# B&R Automation Studio project NAEUL004C00R13L518F00 (part 34)

#### Act_Background3.st - Do Not Change!!!
```iecst
ACTION Act_Background3: //For BHTC Machines

	IF EDGEPOS(tylocalTLBuz.In.bUIManualMod) THEN

		fbBlink(bEn := FALSE);
		fbWarning(bEn := FALSE);

		tylocalTLBuz.Out.bTLRed		:= FALSE;
		tylocalTLBuz.Out.bTLAmber	:= TRUE;
		tylocalTLBuz.Out.bTLGreen	:= FALSE;
		tylocalTLBuz.Out.bBuzBeep	:= FALSE;

	ELSIF tylocalTLBuz.In.bUIManualMod THEN

		IF tylocalTLBuz.In.bErr = TRUE THEN

			fbBlink.tOnTm	:= tylocalTLBuz.In.tTLErrBlinkTm; //Error T#500ms (from NtParam)
			fbBlink.tOffTm	:= tylocalTLBuz.In.tTLErrBlinkTm; //Error T#500ms (from NtParam)

			fbWarning.tOnTm					:= tylocalTLBuz.In.tBuzErrOnTm; //Warn T#500ms (from NtParam)
			fbWarning.tOffTm				:= tylocalTLBuz.In.tBuzErrOnTm; //Warn T#500ms (from NtParam)
			fbWarning.tRstTm				:= tylocalTLBuz.In.tBuzErrRestTm; //Rest 5 seconds (from NtParam)
			fbWarning.usiOnCnt				:= tylocalTLBuz.In.usiBuzErrOnCntr; //Count 3 times (from NtParam)
			fbWarning.bStopAftRptSeqEn		:= tylocalTLBuz.In.bBuzErrStopSeqEn; //Enable Sequence Count (from NtParam)
			fbWarning.usiStopAftRptSeqCntr	:= tylocalTLBuz.In.usiBuzErrStopSeqCntr; //Sequence Counter  (from NtParam)

			fbBlink(bEn := TRUE);
			fbWarning(bEn := TRUE);

			tylocalTLBuz.Out.bTLAmber	:= fbBlink.bOut;
			tylocalTLBuz.Out.bBuzBeep	:= (fbWarning.bOut) AND (tylocalTLBuz.In.bMuteBuz = FALSE);

			bManualErrOn := TRUE;

		ELSIF bManualErrOn THEN

			fbBlink(bEn := FALSE);
			fbWarning(bEn := FALSE);

			tylocalTLBuz.Out.bTLAmber	:= FALSE;
			tylocalTLBuz.Out.bBuzBeep	:= FALSE;

			bManualErrOn := FALSE;

		END_IF

	ELSIF tylocalTLBuz.In.bUIManualMod = FALSE THEN

		bManualErrOn := FALSE;

		IF tylocalTLBuz.In.bStartup = TRUE THEN //Startup, 3 colour ON

			fbBlink(bEn := FALSE);
			fbWarning(bEn := FALSE);

			tylocalTLBuz.Out.bTLBlue		:= TRUE;
			tylocalTLBuz.Out.bTLAmber	:= TRUE;
			tylocalTLBuz.Out.bTLWhite	:= TRUE;
			tylocalTLBuz.Out.bTLGreen	:= TRUE;
			tylocalTLBuz.Out.bBuzBeep	:= FALSE;

		ELSIF tylocalTLBuz.In.bErr = TRUE THEN //Machine Error,Green TL Off, Red TL Blink

			fbBlink.tOnTm	:= tylocalTLBuz.In.tTLErrBlinkTm; //Error T#500ms (from NtParam)
			fbBlink.tOffTm	:= tylocalTLBuz.In.tTLErrBlinkTm; //Error T#500ms (from NtParam)

			fbWarning.tOnTm					:= tylocalTLBuz.In.tBuzErrOnTm; //Warn T#500ms (from NtParam)
			fbWarning.tOffTm				:= tylocalTLBuz.In.tBuzErrOnTm; //Warn T#500ms (from NtParam)
			fbWarning.tRstTm				:= tylocalTLBuz.In.tBuzErrRestTm; //Rest 5 seconds (from NtParam)
			fbWarning.usiOnCnt				:= tylocalTLBuz.In.usiBuzErrOnCntr; //Count 3 times (from NtParam)
			fbWarning.bStopAftRptSeqEn		:= tylocalTLBuz.In.bBuzErrStopSeqEn; //Enable Sequence Count (from NtParam)
			fbWarning.usiStopAftRptSeqCntr	:= tylocalTLBuz.In.usiBuzErrStopSeqCntr; //Sequence Counter  (from NtParam)

			fbBlink(bEn := TRUE);
			fbWarning(bEn := TRUE);

			tylocalTLBuz.Out.bTLBlue		:= FALSE;
			tylocalTLBuz.Out.bTLAmber	:= fbBlink.bOut;
			tylocalTLBuz.Out.bTLWhite	:= FALSE;
			tylocalTLBuz.Out.bTLGreen	:= FALSE;
			tylocalTLBuz.Out.bBuzBeep	:= fbWarning.bOut AND (tylocalTLBuz.In.bMuteBuz = FALSE);

		ELSIF tylocalTLBuz.In.bErrNoBuz = TRUE THEN //not used (Machine Error With No Buz)

			fbBlink.tOnTm	:= tylocalTLBuz.In.tTLErrBlinkTm; //Error T#500ms, not used (from NtParam)
			fbBlink.tOffTm	:= tylocalTLBuz.In.tTLErrBlinkTm; //Error T#500ms, not used (from NtParam)
			fbBlink(bEn := TRUE);
			fbWarning(bEn := FALSE);

			tylocalTLBuz.Out.bTLBlue		:= FALSE;
			tylocalTLBuz.Out.bTLAmber	:= fbBlink.bOut;
			tylocalTLBuz.Out.bTLWhite	:= FALSE;
			tylocalTLBuz.Out.bTLGreen	:= FALSE;
			tylocalTLBuz.Out.bBuzBeep	:= FALSE;

		ELSIF tylocalTLBuz.In.bWarning[0] = TRUE THEN //Warning or AlarmInfo; [Put Conditions in Act_Link.st]

			fbBlink.tOnTm	:= tylocalTLBuz.In.tTLWarnBlinkTm[0]; //Warn T#500ms (from NtParam)
			fbBlink.tOffTm	:= tylocalTLBuz.In.tTLWarnBlinkTm[0]; //Warn T#500ms (from NtParam)

			fbWarning.tOnTm					:= tylocalTLBuz.In.tBuzWarnOnTm[0]; //Warn T#500ms (from NtParam)
			fbWarning.tOffTm				:= tylocalTLBuz.In.tBuzWarnOnTm[0]; //Warn T#500ms (from NtParam)
			fbWarning.tRstTm				:= tylocalTLBuz.In.tBuzWarnRestTm[0]; //Rest 5 seconds (from NtParam)
			fbWarning.usiOnCnt				:= tylocalTLBuz.In.usiBuzWarnOnCntr[0]; //Count 3 times (from NtParam)
			fbWarning.bStopAftRptSeqEn		:= tylocalTLBuz.In.bBuzWarnStopSeqEn[0]; //Enable Sequence Count (from NtParam)
			fbWarning.usiStopAftRptSeqCntr	:= tylocalTLBuz.In.usiBuzWarnStopSeqCntr[0]; //Sequence Counter  (from NtParam)

			fbBlink(bEn := TRUE);
			fbWarning(bEn := TRUE);

			tylocalTLBuz.Out.bTLBlue		:= FALSE;
			tylocalTLBuz.Out.bTLAmber	:= tylocalTLBuz.In.bStandby; //[tylocalTLBuz.In.bStandby ACCESS p_OpsStatusStop], [p_OpsStatusStop	:= ADR(bStatusStop);]
			tylocalTLBuz.Out.bTLWhite	:= fbBlink.bOut;
			tylocalTLBuz.Out.bTLGreen	:= tylocalTLBuz.In.bOps; //[tylocalTLBuz.In.bOps ACCESS p_OpsStatusRun],  [p_OpsStatusRun	:= ADR(bStatusRun)];
			tylocalTLBuz.Out.bBuzBeep	:= fbWarning.bOut AND (tylocalTLBuz.In.bMuteBuz = FALSE);

		ELSIF tylocalTLBuz.In.bStandby = TRUE THEN //not used

			fbBlink.tOnTm	:= tylocalTLBuz.In.tTLWarnBlinkTm[0];
			fbBlink.tOffTm	:= tylocalTLBuz.In.tTLWarnBlinkTm[0];
			fbBlink(bEn := TRUE);
			fbWarning(bEn := FALSE);

			tylocalTLBuz.Out.bTLBlue		:= FALSE;
			tylocalTLBuz.Out.bTLAmber	:= tylocalTLBuz.In.bStandby;
			tylocalTLBuz.Out.bTLWhite	:= fbBlink.bOut;
			tylocalTLBuz.Out.bTLGreen	:= tylocalTLBuz.In.bOps;
			tylocalTLBuz.Out.bBuzBeep	:= FALSE;

		ELSIF tylocalTLBuz.In.bWarning[1] = TRUE THEN //not used

			fbBlink.tOnTm	:= tylocalTLBuz.In.tTLWarnBlinkTm[1];
			fbBlink.tOffTm	:= tylocalTLBuz.In.tTLWarnBlinkTm[1];

			fbWarning.tOnTm					:= tylocalTLBuz.In.tBuzWarnOnTm[1]; //Warn T#500ms (from NtParam)
			fbWarning.tOffTm				:= tylocalTLBuz.In.tBuzWarnOnTm[1]; //Warn T#500ms (from NtParam)
			fbWarning.tRstTm				:= tylocalTLBuz.In.tBuzWarnRestTm[1]; //Rest 5 seconds (from NtParam)
			fbWarning.usiOnCnt				:= tylocalTLBuz.In.usiBuzWarnOnCntr[1]; //Count 3 times (from NtParam)
			fbWarning.bStopAftRptSeqEn		:= tylocalTLBuz.In.bBuzWarnStopSeqEn[1]; //Enable Sequence Count (from NtParam)
			fbWarning.usiStopAftRptSeqCntr	:= tylocalTLBuz.In.usiBuzWarnStopSeqCntr[1]; //Sequence Counter  (from NtParam)

			fbBlink(bEn := TRUE);
			fbWarning(bEn := TRUE);

			tylocalTLBuz.Out.bTLBlue		:= FALSE;
			tylocalTLBuz.Out.bTLAmber	:= tylocalTLBuz.In.bStandby;
			tylocalTLBuz.Out.bTLWhite	:= fbBlink.bOut;
			tylocalTLBuz.Out.bTLGreen	:= tylocalTLBuz.In.bOps;
			tylocalTLBuz.Out.bBuzBeep	:= fbWarning.bOut AND (tylocalTLBuz.In.bMuteBuz = FALSE);

		ELSIF tylocalTLBuz.In.bWarningNoBuz[1] = TRUE THEN //not used

			fbBlink.tOnTm	:= tylocalTLBuz.In.tTLWarnBlinkTm[1];
			fbBlink.tOffTm	:= tylocalTLBuz.In.tTLWarnBlinkTm[1];
			fbBlink(bEn := TRUE);
			fbWarning(bEn := FALSE);

			tylocalTLBuz.Out.bTLBlue		:= FALSE;
			tylocalTLBuz.Out.bTLAmber	:= tylocalTLBuz.In.bStandby;
			tylocalTLBuz.Out.bTLWhite	:= fbBlink.bOut;
			tylocalTLBuz.Out.bTLGreen	:= tylocalTLBuz.In.bOps;
			tylocalTLBuz.Out.bBuzBeep	:= FALSE;

		ELSIF tylocalTLBuz.In.bWarning[2] = TRUE THEN //not used

			fbBlink.tOnTm	:= tylocalTLBuz.In.tTLWarnBlinkTm[2];
			fbBlink.tOffTm	:= tylocalTLBuz.In.tTLWarnBlinkTm[2];

			fbWarning.tOnTm					:= tylocalTLBuz.In.tBuzWarnOnTm[2]; //Warn T#500ms (from NtParam)
			fbWarning.tOffTm				:= tylocalTLBuz.In.tBuzWarnOnTm[2]; //Warn T#500ms (from NtParam)
			fbWarning.tRstTm				:= tylocalTLBuz.In.tBuzWarnRestTm[2]; //Rest 5 seconds (from NtParam)
			fbWarning.usiOnCnt				:= tylocalTLBuz.In.usiBuzWarnOnCntr[2]; //Count 3 times (from NtParam)
			fbWarning.bStopAftRptSeqEn		:= tylocalTLBuz.In.bBuzWarnStopSeqEn[2]; //Enable Sequence Count (from NtParam)
			fbWarning.usiStopAftRptSeqCntr	:= tylocalTLBuz.In.usiBuzWarnStopSeqCntr[2]; //Sequence Counter  (from NtParam)

			fbBlink(bEn := TRUE);
			fbWarning(bEn := TRUE);

			tylocalTLBuz.Out.bTLBlue	:= FALSE;
			tylocalTLBuz.Out.bTLAmber	:= tylocalTLBuz.In.bStandby;
			tylocalTLBuz.Out.bTLWhite	:= fbBlink.bOut;
			tylocalTLBuz.Out.bTLGreen	:= tylocalTLBuz.In.bOps;
			tylocalTLBuz.Out.bBuzBeep	:= fbWarning.bOut AND (tylocalTLBuz.In.bMuteBuz = FALSE);

		ELSIF tylocalTLBuz.In.bWarningNoBuz[2] = TRUE THEN //not used

			fbBlink.tOnTm	:= tylocalTLBuz.In.tTLWarnBlinkTm[2];
			fbBlink.tOffTm	:= tylocalTLBuz.In.tTLWarnBlinkTm[2];
			fbBlink(bEn := TRUE);
			fbWarning(bEn := FALSE);

			tylocalTLBuz.Out.bTLBlue		:= FALSE;
			tylocalTLBuz.Out.bTLAmber	:= tylocalTLBuz.In.bStandby;
			tylocalTLBuz.Out.bTLWhite	:= fbBlink.bOut;
			tylocalTLBuz.Out.bTLGreen	:= tylocalTLBuz.In.bOps;
			tylocalTLBuz.Out.bBuzBeep	:= FALSE;

		ELSIF tylocalTLBuz.In.bWarning[3] = TRUE THEN //not used

			fbBlink.tOnTm	:= tylocalTLBuz.In.tTLWarnBlinkTm[3];
			fbBlink.tOffTm	:= tylocalTLBuz.In.tTLWarnBlinkTm[3];

			fbWarning.tOnTm					:= tylocalTLBuz.In.tBuzWarnOnTm[3]; //Warn T#500ms (from NtParam)
			fbWarning.tOffTm				:= tylocalTLBuz.In.tBuzWarnOnTm[3]; //Warn T#500ms (from NtParam)
			fbWarning.tRstTm				:= tylocalTLBuz.In.tBuzWarnRestTm[3]; //Rest 5 seconds (from NtParam)
			fbWarning.usiOnCnt				:= tylocalTLBuz.In.usiBuzWarnOnCntr[3]; //Count 3 times (from NtParam)
			fbWarning.bStopAftRptSeqEn		:= tylocalTLBuz.In.bBuzWarnStopSeqEn[3]; //Enable Sequence Count (from NtParam)
			fbWarning.usiStopAftRptSeqCntr	:= tylocalTLBuz.In.usiBuzWarnStopSeqCntr[3]; //Sequence Counter  (from NtParam)

			fbBlink(bEn := TRUE);
			fbWarning(bEn := TRUE);

			tylocalTLBuz.Out.bTLBlue		:= FALSE;
			tylocalTLBuz.Out.bTLAmber	:= tylocalTLBuz.In.bStandby;
			tylocalTLBuz.Out.bTLWhite	:= fbBlink.bOut;
			tylocalTLBuz.Out.bTLGreen	:= tylocalTLBuz.In.bOps;
			tylocalTLBuz.Out.bBuzBeep	:= fbWarning.bOut AND (tylocalTLBuz.In.bMuteBuz = FALSE);

		ELSIF tylocalTLBuz.In.bWarningNoBuz[3] = TRUE THEN //not used

			fbBlink.tOnTm	:= tylocalTLBuz.In.tTLWarnBlinkTm[3];
			fbBlink.tOffTm	:= tylocalTLBuz.In.tTLWarnBlinkTm[3];
			fbBlink(bEn := TRUE);
			fbWarning(bEn := FALSE);

			tylocalTLBuz.Out.bTLBlue		:= FALSE;
			tylocalTLBuz.Out.bTLAmber	:= tylocalTLBuz.In.bStandby;
			tylocalTLBuz.Out.bTLWhite	:= fbBlink.bOut;
			tylocalTLBuz.Out.bTLGreen	:= tylocalTLBuz.In.bOps;
			tylocalTLBuz.Out.bBuzBeep	:= FALSE;

		ELSIF tylocalTLBuz.In.bWarning[4] = TRUE THEN //not used

			fbBlink.tOnTm	:= tylocalTLBuz.In.tTLWarnBlinkTm[4];
			fbBlink.tOffTm	:= tylocalTLBuz.In.tTLWarnBlinkTm[4];

			fbWarning.tOnTm					:= tylocalTLBuz.In.tBuzWarnOnTm[4]; //Warn T#500ms (from NtParam)
			fbWarning.tOffTm				:= tylocalTLBuz.In.tBuzWarnOnTm[4]; //Warn T#500ms (from NtParam)
			fbWarning.tRstTm				:= tylocalTLBuz.In.tBuzWarnRestTm[4]; //Rest 5 seconds (from NtParam)
			fbWarning.usiOnCnt				:= tylocalTLBuz.In.usiBuzWarnOnCntr[4]; //Count 3 times (from NtParam)
			fbWarning.bStopAftRptSeqEn		:= tylocalTLBuz.In.bBuzWarnStopSeqEn[4]; //Enable Sequence Count (from NtParam)
			fbWarning.usiStopAftRptSeqCntr	:= tylocalTLBuz.In.usiBuzWarnStopSeqCntr[4]; //Sequence Counter  (from NtParam)

			fbBlink(bEn := TRUE);
			fbWarning(bEn := TRUE);

			tylocalTLBuz.Out.bTLBlue		:= FALSE;
			tylocalTLBuz.Out.bTLAmber	:= tylocalTLBuz.In.bStandby;
			tylocalTLBuz.Out.bTLWhite	:= fbBlink.bOut;
			tylocalTLBuz.Out.bTLGreen	:= tylocalTLBuz.In.bOps;
			tylocalTLBuz.Out.bBuzBeep	:= fbWarning.bOut AND (tylocalTLBuz.In.bMuteBuz = FALSE);

		ELSIF tylocalTLBuz.In.bWarningNoBuz[4] = TRUE THEN //not used

			fbBlink.tOnTm	:= tylocalTLBuz.In.tTLWarnBlinkTm[4];
			fbBlink.tOffTm	:= tylocalTLBuz.In.tTLWarnBlinkTm[4];
			fbBlink(bEn := TRUE);
			fbWarning(bEn := FALSE);

			tylocalTLBuz.Out.bTLBlue		:= FALSE;
			tylocalTLBuz.Out.bTLAmber	:= tylocalTLBuz.In.bStandby;
			tylocalTLBuz.Out.bTLWhite	:= fbBlink.bOut;
			tylocalTLBuz.Out.bTLGreen	:= tylocalTLBuz.In.bOps;
			tylocalTLBuz.Out.bBuzBeep	:= FALSE;

		ELSIF tylocalTLBuz.In.bWarning[5] = TRUE THEN //not used

			fbBlink.tOnTm	:= tylocalTLBuz.In.tTLWarnBlinkTm[5];
			fbBlink.tOffTm	:= tylocalTLBuz.In.tTLWarnBlinkTm[5];

			fbWarning.tOnTm					:= tylocalTLBuz.In.tBuzWarnOnTm[5]; //Warn T#500ms (from NtParam)
			fbWarning.tOffTm				:= tylocalTLBuz.In.tBuzWarnOnTm[5]; //Warn T#500ms (from NtParam)
			fbWarning.tRstTm				:= tylocalTLBuz.In.tBuzWarnRestTm[5]; //Rest 5 seconds (from NtParam)
			fbWarning.usiOnCnt				:= tylocalTLBuz.In.usiBuzWarnOnCntr[5]; //Count 3 times (from NtParam)
			fbWarning.bStopAftRptSeqEn		:= tylocalTLBuz.In.bBuzWarnStopSeqEn[5]; //Enable Sequence Count (from NtParam)
			fbWarning.usiStopAftRptSeqCntr	:= tylocalTLBuz.In.usiBuzWarnStopSeqCntr[5]; //Sequence Counter  (from NtParam)

			fbBlink(bEn := TRUE);
			fbWarning(bEn := TRUE);

			tylocalTLBuz.Out.bTLBlue		:= FALSE;
			tylocalTLBuz.Out.bTLAmber	:= tylocalTLBuz.In.bStandby;
			tylocalTLBuz.Out.bTLWhite	:= fbBlink.bOut;
			tylocalTLBuz.Out.bTLGreen	:= tylocalTLBuz.In.bOps;
			tylocalTLBuz.Out.bBuzBeep	:= fbWarning.bOut AND (tylocalTLBuz.In.bMuteBuz = FALSE);

		ELSIF tylocalTLBuz.In.bWarningNoBuz[5] = TRUE THEN //not used

			fbBlink.tOnTm	:= tylocalTLBuz.In.tTLWarnBlinkTm[5];
			fbBlink.tOffTm	:= tylocalTLBuz.In.tTLWarnBlinkTm[5];
			fbBlink(bEn := TRUE);
			fbWarning(bEn := FALSE);

			tylocalTLBuz.Out.bTLBlue		:= FALSE;
			tylocalTLBuz.Out.bTLAmber	:= tylocalTLBuz.In.bStandby;
			tylocalTLBuz.Out.bTLWhite	:= fbBlink.bOut;
			tylocalTLBuz.Out.bTLGreen	:= tylocalTLBuz.In.bOps;
			tylocalTLBuz.Out.bBuzBeep	:= FALSE;

		ELSIF tylocalTLBuz.In.bSeqStop = TRUE THEN //[p_bSeqStop ACCESS p_OpsStatusCycleStop] ,[p_OpsStatusCycleStop	:= ADR(bStatusCycleStop);]

			fbBlink.tOnTm	:= tBlinkTm; //Local T#500ms
			fbBlink.tOffTm	:= tBlinkTm; //Local T#500ms
			fbBlink(bEn := TRUE);
			fbWarning(bEn := FALSE);

			tylocalTLBuz.Out.bTLBlue		:= FALSE;
			tylocalTLBuz.Out.bTLAmber	:= fbBlink.bOut;
			tylocalTLBuz.Out.bTLWhite	:= FALSE;
			tylocalTLBuz.Out.bTLGreen	:= TRUE;
			tylocalTLBuz.Out.bBuzBeep	:= FALSE;

		ELSIF tylocalTLBuz.In.bChgRcp = TRUE THEN //Change Rcp, Disco Light, not used

			fbBlink.tOnTm	:= tylocalTLBuz.In.tTLChgRcpBlinkTm; //Chg Rcp T#500ms (from NtParam)
			fbBlink.tOffTm	:= tylocalTLBuz.In.tTLChgRcpBlinkTm; //Chg Rcp T#500ms (from NtParam)
			fbBlink(bEn := TRUE);
			fbWarning(bEn := FALSE);

			IF EDGE(fbBlink.bOut) THEN
				IF tylocalTLBuz.Out.bTLAmber = TRUE THEN
					tylocalTLBuz.Out.bTLAmber	:= FALSE;
					tylocalTLBuz.Out.bTLWhite	:= FALSE;
					tylocalTLBuz.Out.bTLGreen	:= TRUE;
				ELSIF tylocalTLBuz.Out.bTLWhite = TRUE THEN
					tylocalTLBuz.Out.bTLAmber	:= TRUE;
					tylocalTLBuz.Out.bTLWhite	:= FALSE;
					tylocalTLBuz.Out.bTLGreen	:= FALSE;
				ELSE
					tylocalTLBuz.Out.bTLAmber	:= FALSE;
					tylocalTLBuz.Out.bTLWhite	:= TRUE;
					tylocalTLBuz.Out.bTLGreen	:= FALSE;
				END_IF
			END_IF

			tylocalTLBuz.Out.bBuzBeep	:= fbBlink.bOut AND (tylocalTLBuz.In.bMuteBuz = FALSE);

		ELSIF tylocalTLBuz.In.bStep = TRUE THEN //not used, [p_bStep ACCESS p_OpsStatusStep], [p_OpsStatusStep	:= ADR(bStatusStep);]

			fbBlink.tOnTm	:= tBlinkTm;
			fbBlink.tOffTm	:= tBlinkTm;
			fbBlink(bEn := TRUE);
			fbWarning(bEn := FALSE);

			tylocalTLBuz.Out.bTLBlue		:= FALSE;
			tylocalTLBuz.Out.bTLAmber	:= FALSE;
			tylocalTLBuz.Out.bTLWhite	:= FALSE;
			tylocalTLBuz.Out.bTLGreen	:= fbBlink.bOut;
			tylocalTLBuz.Out.bBuzBeep	:= FALSE;

		ELSIF tylocalTLBuz.In.bOps = TRUE THEN //Auto Mode, Green TL only

			fbBlink(bEn := FALSE);
			fbWarning(bEn := FALSE);

			tylocalTLBuz.Out.bTLRed		:= FALSE;
			tylocalTLBuz.Out.bTLAmber	:= FALSE;
			tylocalTLBuz.Out.bTLGreen	:= TRUE;
			tylocalTLBuz.Out.bBuzBeep	:= FALSE;

		ELSIF tylocalTLBuz.In.bSimulation = TRUE THEN //For simulation

			fbBlink.tOnTm	:= tBlinkTm;
			fbBlink.tOffTm	:= tBlinkTm;
			fbBlink(bEn := TRUE);
			fbWarning(bEn := FALSE);

			tylocalTLBuz.Out.bTLBlue		:= fbBlink.bOut;
			tylocalTLBuz.Out.bTLAmber	:= fbBlink.bOut;
			tylocalTLBuz.Out.bTLWhite	:= fbBlink.bOut;
			tylocalTLBuz.Out.bTLGreen	:= TRUE;
			tylocalTLBuz.Out.bBuzBeep	:= FALSE;

		ELSIF tylocalTLBuz.In.bStandby = TRUE THEN //Stop Mode, On Red TL only

			fbBlink(bEn := FALSE);
			fbWarning(bEn := FALSE);

			tylocalTLBuz.Out.bTLBlue		:= FALSE;
			tylocalTLBuz.Out.bTLAmber	:= TRUE;
			tylocalTLBuz.Out.bTLWhite	:= FALSE;
			tylocalTLBuz.Out.bTLGreen	:= FALSE;
			tylocalTLBuz.Out.bBuzBeep	:= FALSE;

		ELSE //Resest if nothing else

			fbBlink(bEn := FALSE);
			fbWarning(bEn := FALSE);

			tylocalTLBuz.Out.bTLBlue		:= FALSE;
			tylocalTLBuz.Out.bTLAmber	:= FALSE;
			tylocalTLBuz.Out.bTLWhite	:= FALSE;
			tylocalTLBuz.Out.bTLGreen	:= FALSE;
			tylocalTLBuz.Out.bBuzBeep	:= FALSE;

		END_IF

	END_IF

	IF tylocalTLBuz.In.bUIManualMod = FALSE AND tylocalTLBuz.In.bErr = FALSE THEN
		IF tylocalTLBuz.In.bTLAmberFlashEn THEN //Amber Flash 1 sec [Put Conditions in Act_Link.st]

			fbBlink1.tOnTm	:= tylocalTLBuz.In.tTLAmberBlinkTm; //T#500ms (from NtParam)
			fbBlink1.tOffTm	:= tylocalTLBuz.In.tTLAmberBlinkTm; //T#500ms (from NtParam)
			fbBlink1(bEn := TRUE);

			tylocalTLBuz.Out.bTLAmber	:= fbBlink1.bOut;

		ELSE
			fbBlink1(bEn := FALSE);
		END_IF

		IF tylocalTLBuz.In.bTLWhiteFlashEn THEN //White Flash 1 sec [Put Conditions in Act_Link.st]

			fbBlink2.tOnTm	:= tylocalTLBuz.In.tTLWhiteBlinkTm; //T#500ms (from NtParam)
			fbBlink2.tOffTm	:= tylocalTLBuz.In.tTLWhiteBlinkTm; //T#500ms (from NtParam)
			fbBlink2(bEn := TRUE);

			tylocalTLBuz.Out.bTLWhite		:= fbBlink2.bOut;
		ELSE
			fbBlink2(bEn := FALSE);
		END_IF

		IF tylocalTLBuz.In.bTLGreenFlashEn THEN //Green Flash 1 sec [Put Conditions in Act_Link.st]

			fbBlink3.tOnTm	:= tylocalTLBuz.In.tTLGreenBlinkTm; //T#500ms (from NtParam)
			fbBlink3.tOffTm	:= tylocalTLBuz.In.tTLGreenBlinkTm; //T#500ms (from NtParam)
			fbBlink3(bEn := TRUE);

			tylocalTLBuz.Out.bTLGreen	:= fbBlink3.bOut;
		ELSE
			fbBlink3(bEn := FALSE);
		END_IF

		IF tylocalTLBuz.In.bTLBlueFlashEn THEN //Blue Flash 1 sec [Put Conditions in Act_Link.st]

			fbBlink4.tOnTm	:= tylocalTLBuz.In.tTLBlueBlinkTm; //T#500ms (from NtParam)
			fbBlink4.tOffTm	:= tylocalTLBuz.In.tTLBlueBlinkTm; //T#500ms (from NtParam)
			fbBlink4(bEn := TRUE);

			tylocalTLBuz.Out.bTLGreen	:= fbBlink4.bOut;
		ELSE
			fbBlink4(bEn := FALSE);
		END_IF

		IF tylocalTLBuz.In.bBuzAlertEn = TRUE AND fbWarning.bEn=FALSE THEN

			fbWarning1.tOnTm				:= tylocalTLBuz.In.tBuzAlertOnTm;
			fbWarning1.tOffTm				:= tylocalTLBuz.In.tBuzAlertOnTm;
			fbWarning1.tRstTm				:= tylocalTLBuz.In.tBuzAlertRestTm;
			fbWarning1.usiOnCnt				:= tylocalTLBuz.In.usiBuzAlertOnCntr;
			fbWarning1.bStopAftRptSeqEn		:= tylocalTLBuz.In.bBuzAlertStopSeqEn; //Enable Sequence Count (from NtParam)
			fbWarning1.usiStopAftRptSeqCntr	:= tylocalTLBuz.In.usiBuzAlertStopSeqCntr; //Sequence Counter  (from NtParam)

			fbWarning1(bEn := TRUE);

			tylocalTLBuz.Out.bBuzBeep	:= fbWarning1.bOut AND (tylocalTLBuz.In.bMuteBuz = FALSE);

		ELSE
			fbWarning1(bEn := FALSE);
		END_IF
	ELSE
		fbBlink1(bEn := FALSE);
		fbBlink2(bEn := FALSE);
		fbBlink3(bEn := FALSE);
		fbBlink4(bEn := FALSE);
		fbWarning1(bEn := FALSE);
	END_IF

	//Arrange tylocalTLBuz.In.bWarning according to the severity of the warning or info (Err is prioritized)
	IF tylocalTLBuz.In.bErr THEN
		usiWarnInfoStateNew	:= 1;
	ELSIF tylocalTLBuz.In.bWarning[0] THEN
		usiWarnInfoStateNew	:= 2;
	ELSIF tylocalTLBuz.In.bWarning[1] THEN
		usiWarnInfoStateNew	:= 3;
	ELSIF tylocalTLBuz.In.bWarning[2] THEN
		usiWarnInfoStateNew	:= 4;
	ELSIF tylocalTLBuz.In.bWarning[3] THEN
		usiWarnInfoStateNew	:= 5;
	ELSIF tylocalTLBuz.In.bWarning[4] THEN
		usiWarnInfoStateNew	:= 6;
	ELSIF tylocalTLBuz.In.bWarning[5] THEN
		usiWarnInfoStateNew	:= 7;
	ELSIF tylocalTLBuz.In.bBuzAlertEn AND fbWarning.bEn=FALSE THEN
		usiWarnInfoStateNew	:= 8;
	ELSE
		usiWarnInfoStateNew	:= 0;
	END_IF

	IF usiWarnInfoStateOld<>usiWarnInfoStateNew THEN
		usiWarnInfoStateOld:=usiWarnInfoStateNew;
		fbWarning(bEn := FALSE);
		fbWarning1(bEn := FALSE);
	END_IF

END_ACTION
```

#### Act_Background4.st - Do Not Change!!!
```iecst
ACTION Act_Background4:

	IF EDGEPOS(tylocalTLBuz.In.bUIManualMod) THEN

		fbBlink(bEn := FALSE);
		fbWarning(bEn := FALSE);

		tylocalTLBuz.In.bTLRed		:= FALSE;
		tylocalTLBuz.In.bTLAmber	:= TRUE;
		tylocalTLBuz.In.bTLWhite	:= TRUE;
		tylocalTLBuz.In.bTLGreen	:= FALSE;
		tylocalTLBuz.In.bBuzBeep	:= FALSE;

	ELSIF tylocalTLBuz.In.bUIManualMod THEN

		IF tylocalTLBuz.In.bErr = TRUE THEN

			fbBlink.tOnTm	:= tylocalTLBuz.In.tTLErrBlinkTm; //Error T#500ms (from NtParam)
			fbBlink.tOffTm	:= tylocalTLBuz.In.tTLErrBlinkTm; //Error T#500ms (from NtParam)

			fbWarning.tOnTm					:= p_tBuzErrOnTm; //Warn T#500ms (from NtParam)
			fbWarning.tOffTm				:= p_tBuzErrOnTm; //Warn T#500ms (from NtParam)
			fbWarning.tRstTm				:= p_tBuzErrRestTm; //Rest 5 seconds (from NtParam)
			fbWarning.usiOnCnt				:= p_usiBuzErrOnCntr; //Count 3 times (from NtParam)
			fbWarning.bStopAftRptSeqEn		:= p_bBuzErrStopSeqEn; //Enable Sequence Count (from NtParam)
			fbWarning.usiStopAftRptSeqCntr	:= p_usiBuzErrStopSeqCntr; //Sequence Counter  (from NtParam)

			fbBlink(bEn := TRUE);
			fbWarning(bEn := TRUE);

			tylocalTLBuz.In.bTLRed		:= fbBlink.bOut;
			tylocalTLBuz.In.bBuzBeep	:= (fbWarning.bOut) AND (p_bMuteBuz = FALSE);

			bManualErrOn := TRUE;
			tylocalTLBuz.In.bBuzAlertEn := FALSE;

		ELSIF bManualErrOn THEN

			fbBlink(bEn := FALSE);
			fbWarning(bEn := FALSE);

			tylocalTLBuz.In.bTLRed		:= FALSE;
			tylocalTLBuz.In.bBuzBeep	:= FALSE;

			bManualErrOn := FALSE;
			tylocalTLBuz.In.bBuzAlertEn := FALSE;

		END_IF
	ELSIF p_bManual = FALSE THEN

		bManualErrOn := FALSE;
		IF p_bStartup THEN
			tylocalTLBuz.In.bTLGreen := FALSE;
			tylocalTLBuz.In.bTLWhite := FALSE;
			tylocalTLBuz.In.bTLGreenFlashEn := TRUE;
			tylocalTLBuz.In.bTLWhiteFlashEn := TRUE;
			tylocalTLBuz.In.bBuzBeep := FALSE;
			tylocalTLBuz.In.bBuzAlertEn := FALSE;

		ELSIF p_bOps THEN
			tylocalTLBuz.In.bTLGreen := TRUE;
			tylocalTLBuz.In.bTLWhite := FALSE;
			tylocalTLBuz.In.bTLGreenFlashEn := FALSE;
			tylocalTLBuz.In.bTLWhiteFlashEn := FALSE;
			tylocalTLBuz.In.bBuzBeep := FALSE;
			tylocalTLBuz.In.bBuzAlertEn := FALSE;

		ELSIF p_bSeqStop THEN
			tylocalTLBuz.In.bTLGreen := FALSE;
			tylocalTLBuz.In.bTLWhite := FALSE;
			tylocalTLBuz.In.bTLGreenFlashEn := TRUE;
			tylocalTLBuz.In.bTLWhiteFlashEn := FALSE;
			tylocalTLBuz.In.bBuzBeep := FALSE;
			tylocalTLBuz.In.bBuzAlertEn := FALSE;

		ELSIF p_bStandby THEN
			tylocalTLBuz.In.bTLGreen := FALSE;
			tylocalTLBuz.In.bTLWhite := FALSE;
			tylocalTLBuz.In.bTLGreenFlashEn := FALSE;
			tylocalTLBuz.In.bTLWhiteFlashEn := TRUE;
			tylocalTLBuz.In.bBuzBeep := FALSE;
			tylocalTLBuz.In.bBuzAlertEn := FALSE;

		ELSIF p_bSimulation THEN
			tylocalTLBuz.In.bTLGreen := TRUE;
			tylocalTLBuz.In.bTLWhite := FALSE;
			tylocalTLBuz.In.bTLGreenFlashEn := FALSE;
			tylocalTLBuz.In.bTLWhiteFlashEn := TRUE;
			tylocalTLBuz.In.bBuzBeep := FALSE;
			tylocalTLBuz.In.bBuzAlertEn := FALSE;

		END_IF

		bFullMag :=(g_tyBuffer1.tyBffrStat.bBffrFull OR g_tyBuffer2.tyBffrStat.bBffrFull OR g_tyBuffer3.tyBffrStat.bBffrFull);
		IF g_tyMcParamCurr.bAGVComEn THEN

			IF bFullMag THEN
//				tylocalTLBuz.In.bTLGreen := FALSE;
				tylocalTLBuz.In.bTLWhite := FALSE;
				tylocalTLBuz.In.bTLGreenFlashEn := FALSE;
				tylocalTLBuz.In.bTLWhiteFlashEn := TRUE;
				tylocalTLBuz.In.bBuzBeep := FALSE;
				tylocalTLBuz.In.bBuzAlertEn := FALSE;
			END_IF

		END_IF

		IF tylocalTLBuz.In.bWarning[0] THEN
			IF p_bOps THEN
				tylocalTLBuz.In.bTLGreen := TRUE;
				tylocalTLBuz.In.bTLWhite := FALSE;
				tylocalTLBuz.In.bTLGreenFlashEn := FALSE;
				tylocalTLBuz.In.bTLWhiteFlashEn := TRUE;
			ELSIF p_bSeqStop THEN
				tylocalTLBuz.In.bTLGreen := FALSE;
				tylocalTLBuz.In.bTLWhite := FALSE;
				tylocalTLBuz.In.bTLGreenFlashEn := TRUE;
				tylocalTLBuz.In.bTLWhiteFlashEn := TRUE;
			ELSE
				tylocalTLBuz.In.bTLGreen := FALSE;
				tylocalTLBuz.In.bTLWhite := FALSE;
				tylocalTLBuz.In.bTLGreenFlashEn := FALSE;
				tylocalTLBuz.In.bTLWhiteFlashEn := TRUE;
			END_IF

			IF p_eMcParamMagExMode = McSetMagXcAutoMode THEN //p_bMcParamAGVComEn
				tylocalTLBuz.In.bBuzAlertEn := FALSE;
			ELSE
				tylocalTLBuz.In.bBuzAlertEn := TRUE;
			END_IF
//			IF tylocalTLBuz.In.bBuzBeep = TRUE AND p_bMcParamAGVComEn AND bFullMag THEN
//				tylocalTLBuz.In.bBuzBeep := FALSE;
//			ELSE
//				tylocalTLBuz.In.bBuzBeep := TRUE;
//			END_IF
//			tylocalTLBuz.In.bBuzAlertEn := TRUE;
		END_IF

		IF tylocalTLBuz.In.bErr THEN
			fbBlink.tOnTm	:= tylocalTLBuz.In.tTLErrBlinkTm; //Error T#500ms (from NtParam)
			fbBlink.tOffTm	:= tylocalTLBuz.In.tTLErrBlinkTm; //Error T#500ms (from NtParam)

			fbWarning.tOnTm					:= p_tBuzErrOnTm; //Warn T#500ms (from NtParam)
			fbWarning.tOffTm				:= p_tBuzErrOnTm; //Warn T#500ms (from NtParam)
			fbWarning.tRstTm				:= p_tBuzErrRestTm; //Rest 5 seconds (from NtParam)
			fbWarning.usiOnCnt				:= p_usiBuzErrOnCntr; //Count 3 times (from NtParam)
			fbWarning.bStopAftRptSeqEn		:= p_bBuzErrStopSeqEn; //Enable Sequence Count (from NtParam)
			fbWarning.usiStopAftRptSeqCntr	:= p_usiBuzErrStopSeqCntr; //Sequence Counter  (from NtParam)

			fbBlink(bEn := TRUE);
			fbWarning(bEn := TRUE);

			tylocalTLBuz.In.bTLRed		:= fbBlink.bOut;
			tylocalTLBuz.In.bTLAmber	:= FALSE;
			tylocalTLBuz.In.bTLGreen	:= FALSE;
			tylocalTLBuz.In.bBuzBeep	:= (fbWarning.bOut) AND (p_bMuteBuz = FALSE);
			tylocalTLBuz.In.bBuzAlertEn := FALSE;
		END_IF

		IF tylocalTLBuz.In.bTLWhiteFlashEn THEN //White Flash 1 sec [Put Conditions in Act_Link.st]

			fbBlink2.tOnTm	:= p_tTLWhiteBlinkTm; //T#500ms (from NtParam)
			fbBlink2.tOffTm	:= p_tTLWhiteBlinkTm; //T#500ms (from NtParam)
			fbBlink2(bEn := TRUE);

			tylocalTLBuz.In.bTLWhite		:= fbBlink2.bOut;
		ELSE
			fbBlink2(bEn := FALSE);
		END_IF

		IF tylocalTLBuz.In.bTLGreenFlashEn THEN //Green Flash 1 sec [Put Conditions in Act_Link.st]

			fbBlink3.tOnTm	:= p_tTLGreenBlinkTm; //T#500ms (from NtParam)
			fbBlink3.tOffTm	:= p_tTLGreenBlinkTm; //T#500ms (from NtParam)
			fbBlink3(bEn := TRUE);

			tylocalTLBuz.In.bTLGreen	:= fbBlink3.bOut;
		ELSE
			fbBlink3(bEn := FALSE);
		END_IF

		IF tylocalTLBuz.In.bBuzAlertEn THEN

			fbWarning1.tOnTm				:= p_tBuzAlertOnTm;
			fbWarning1.tOffTm				:= p_tBuzAlertOnTm;
			fbWarning1.tRstTm				:= p_tBuzAlertRestTm;
			fbWarning1.usiOnCnt				:= p_usiBuzAlertOnCntr;
			fbWarning1.bStopAftRptSeqEn		:= p_bBuzAlertStopSeqEn; //Enable Sequence Count (from NtParam)
			fbWarning1.usiStopAftRptSeqCntr	:= p_usiBuzAlertStopSeqCntr; //Sequence Counter  (from NtParam)

			fbWarning1(bEn := TRUE);

			tylocalTLBuz.In.bBuzBeep	:= fbWarning1.bOut AND (p_bMuteBuz = FALSE);

		ELSE
			fbWarning1(bEn := FALSE);
		END_IF
	END_IF

END_ACTION
```

#### Local.var - Do Not Change!!!
```iecst
(*2020-03-16*)
VAR
	tylocalTLBuz : tyTLBuz;
END_VAR
(**)
(*Local Action, State & Status*)
VAR
	eAct : eTLBuzAction := TLBuzActIdle;
	eStat : eTLBuzAction := TLBuzActIdle;
	eStatus : eFBStatus := Idle;
	sStatTxt : STRING[200] := '';
	a_sStatText : ARRAY[0..50] OF STRING[200] := ['Idling','Turning On Tower Light Green','Turning On Tower Light Amber','Turning On Tower Light Red','Turning On Buzzer','Turning Off Tower Light Green','Turning Off Tower Light Amber','Turning Off Tower Light Red','Turning Off Buzzer','Turning On All Output','Turning Off All Output',40('')];
END_VAR
(**)
(*Local Alarm*)
(**)
(*Local Output*)
VAR
	bTLBlue : BOOL;
	bTLRed : BOOL;
	bTLAmber : BOOL;
	bTLWhite : BOOL;
	bTLGreen : BOOL;
	bBuzBeep : BOOL;
END_VAR
(**)
(*Local Input*)
VAR
	bManualErrOn : BOOL := FALSE;
	bManual : BOOL := FALSE;
	bStartup : BOOL := FALSE;
	bErr : BOOL := FALSE;
	bErrNoBuz : BOOL := FALSE;
	bWarning : BOOL := FALSE;
	bWarningNoBuz : BOOL := FALSE;
	bWarning1 : BOOL := FALSE;
	bWarning1NoBuz : BOOL := FALSE;
	bWarning2 : BOOL := FALSE;
	bWarning2NoBuz : BOOL := FALSE;
	bWarning3 : BOOL := FALSE;
	bWarning3NoBuz : BOOL := FALSE;
	bWarning4 : BOOL := FALSE;
	bWarning4NoBuz : BOOL := FALSE;
	bWarning5 : BOOL := FALSE;
	bWarning5NoBuz : BOOL := FALSE;
	bChgRcp : BOOL := FALSE;
	bSeqStop : BOOL := FALSE;
	bStep : BOOL := FALSE;
	bOps : BOOL := FALSE;
	bStandby : BOOL := FALSE;
	bSimulation : BOOL := FALSE;
	bMuteBuz : BOOL := FALSE;
	tTLChgRcpBlinkTm : TIME := T#200ms;
	tTLErrBlinkTm : TIME := T#500ms;
	tBuzErrOnTm : TIME := T#500ms;
	tBuzErrRestTm : TIME := T#500ms;
	usiBuzErrOnCntr : USINT := 3;
	bBuzErrStopSeqEn : BOOL := FALSE;
	usiBuzErrStopSeqCntr : USINT := 3;
	tTLWarnBlinkTm : TIME := T#500ms;
	tBuzWarnOnTm : TIME := T#500ms;
	tBuzWarnRestTm : TIME := T#5s;
	usiBuzWarnOnCntr : USINT := 3;
	bBuzWarnStopSeqEn : BOOL := FALSE;
	usiBuzWarnStopSeqCntr : USINT := 3;
	tTLWarn1BlinkTm : TIME := T#500ms;
	tBuzWarn1OnTm : TIME := T#500ms;
	tBuzWarn1RestTm : TIME := T#5s;
	usiBuzWarn1OnCntr : USINT := 3;
	bBuzWarn1StopSeqEn : BOOL := FALSE;
	usiBuzWarn1StopSeqCntr : USINT := 3;
	tTLWarn2BlinkTm : TIME := T#500ms;
	tBuzWarn2OnTm : TIME := T#500ms;
	tBuzWarn2RestTm : TIME := T#5s;
	usiBuzWarn2OnCntr : USINT := 3;
	bBuzWarn2StopSeqEn : BOOL := FALSE;
	usiBuzWarn2StopSeqCntr : USINT := 3;
	tTLWarn3BlinkTm : TIME := T#500ms;
	tBuzWarn3OnTm : TIME := T#500ms;
	tBuzWarn3RestTm : TIME := T#5s;
	usiBuzWarn3OnCntr : USINT := 3;
	bBuzWarn3StopSeqEn : BOOL := FALSE;
	usiBuzWarn3StopSeqCntr : USINT := 3;
	tTLWarn4BlinkTm : TIME := T#500ms;
	tBuzWarn4OnTm : TIME := T#500ms;
	tBuzWarn4RestTm : TIME := T#5s;
	usiBuzWarn4OnCntr : USINT := 3;
	bBuzWarn4StopSeqEn : BOOL := FALSE;
	usiBuzWarn4StopSeqCntr : USINT := 3;
	tTLWarn5BlinkTm : TIME := T#500ms;
	tBuzWarn5OnTm : TIME := T#500ms;
	tBuzWarn5RestTm : TIME := T#5s;
	usiBuzWarn5OnCntr : USINT := 3;
	bBuzWarn5StopSeqEn : BOOL := FALSE;
	usiBuzWarn5StopSeqCntr : USINT := 3;
	tBuzAlertOnTm : TIME := T#500ms;
	tBuzAlertRestTm : TIME := T#5s;
	usiBuzAlertOnCntr : USINT := 3;
	bBuzAlertStopSeqEn : BOOL := FALSE;
	usiBuzAlertStopSeqCntr : USINT := 3;
	tTLBlueBlinkTm : TIME := T#500ms;
	tTLAmberBlinkTm : TIME := T#500ms;
	tTLWhiteBlinkTm : TIME := T#500ms;
	tTLRedBlinkTm : TIME := T#500ms;
	tTLGreenBlinkTm : TIME := T#500ms;
	bCoveSwitchSig : BOOL := FALSE;
	eTLBuzMode : eTLBuzMod := TLBuzModNutek;
	bAOIErrSig : BOOL := FALSE;
	bAOIOriginSig : BOOL := FALSE;
	bBuzAlertEn : BOOL := FALSE;
	bTLBlueFlashEn : BOOL := FALSE;
	bTLAmberFlashEn : BOOL := FALSE;
	bTLWhiteFlashEn : BOOL := FALSE;
	bTLRedFlashEn : BOOL := FALSE;
	bTLGreenFlashEn : BOOL := FALSE;
	bFullMag : BOOL;
END_VAR
(**)
(*Local*)
VAR
	usiWarnInfoStateOld : USINT; (*Default buzzer behavior*)
	usiWarnInfoStateNew : USINT; (*Default buzzer behavior*)
	bInitDone : BOOL;
	bInitialDone : BOOL;
	tBlinkTm : TIME := T#500ms;
	fbBlink : fbTLBuzBlink;
	fbBlink1 : fbTLBuzBlink;
	fbBlink2 : fbTLBuzBlink;
	fbBlink3 : fbTLBuzBlink;
	fbBlink4 : fbTLBuzBlink;
	fbWarning : fbTLBuzWarn;
	fbWarning1 : fbTLBuzWarn;
	eStatOld : eTLBuzAction := TLBuzActIdle;
END_VAR
```

#### InputRef.var - not listed in the package file held
```iecst
(*2020-03-16*)
(**)
(*General*)
VAR
	p_eAct : REFERENCE TO eTLBuzAction;
END_VAR
(**)
(*Configuration*)
VAR
	p_bManual : REFERENCE TO BOOL;
	p_bStartup : REFERENCE TO BOOL;
	p_bErr : REFERENCE TO BOOL;
	p_bErrNoBuz : REFERENCE TO BOOL;
	p_bWarning : REFERENCE TO BOOL;
	p_bWarningNoBuz : REFERENCE TO BOOL;
	p_bWarning1 : REFERENCE TO BOOL;
	p_bWarning1NoBuz : REFERENCE TO BOOL;
	p_bWarning2 : REFERENCE TO BOOL;
	p_bWarning2NoBuz : REFERENCE TO BOOL;
	p_bWarning3 : REFERENCE TO BOOL;
	p_bWarning3NoBuz : REFERENCE TO BOOL;
	p_bWarning4 : REFERENCE TO BOOL;
	p_bWarning4NoBuz : REFERENCE TO BOOL;
	p_bWarning5 : REFERENCE TO BOOL;
	p_bWarning5NoBuz : REFERENCE TO BOOL;
	p_bChgRcp : REFERENCE TO BOOL;
	p_bSeqStop : REFERENCE TO BOOL;
	p_bStep : REFERENCE TO BOOL;
	p_bOps : REFERENCE TO BOOL;
	p_bStandby : REFERENCE TO BOOL;
	p_bSimulation : REFERENCE TO BOOL;
	p_bMuteBuz : REFERENCE TO BOOL;
END_VAR
(*TLBuz ChangeRcp Behaviour*)
VAR
	p_tTLChgRcpBlinkTm : REFERENCE TO TIME;
END_VAR
(*TLBuz Error Behaviour*)
VAR
	p_tTLErrBlinkTm : REFERENCE TO TIME;
	p_tBuzErrOnTm : REFERENCE TO TIME;
	p_tBuzErrRestTm : REFERENCE TO TIME;
	p_usiBuzErrOnCntr : REFERENCE TO USINT;
	p_bBuzErrStopSeqEn : REFERENCE TO BOOL;
	p_usiBuzErrStopSeqCntr : REFERENCE TO USINT;
END_VAR
(*TLBuz Default Warning Behaviour*)
VAR
	p_tTLWarnBlinkTm : REFERENCE TO TIME;
	p_tBuzWarnOnTm : REFERENCE TO TIME;
	p_tBuzWarnRestTm : REFERENCE TO TIME;
	p_usiBuzWarnOnCntr : REFERENCE TO USINT;
	p_bBuzWarnStopSeqEn : REFERENCE TO BOOL;
	p_usiBuzWarnStopSeqCntr : REFERENCE TO USINT;
END_VAR
(*TLBuz Special Warning 1 Behaviour*)
VAR
	p_tTLWarn1BlinkTm : REFERENCE TO TIME;
	p_tBuzWarn1OnTm : REFERENCE TO TIME;
	p_tBuzWarn1RestTm : REFERENCE TO TIME;
	p_usiBuzWarn1OnCntr : REFERENCE TO USINT;
	p_bBuzWarn1StopSeqEn : REFERENCE TO BOOL;
	p_usiBuzWarn1StopSeqCntr : REFERENCE TO USINT;
END_VAR
(*TLBuz Special Warning 2 Behaviour*)
VAR
	p_tTLWarn2BlinkTm : REFERENCE TO TIME;
	p_tBuzWarn2OnTm : REFERENCE TO TIME;
	p_tBuzWarn2RestTm : REFERENCE TO TIME;
	p_usiBuzWarn2OnCntr : REFERENCE TO USINT;
	p_bBuzWarn2StopSeqEn : REFERENCE TO BOOL;
	p_usiBuzWarn2StopSeqCntr : REFERENCE TO USINT;
END_VAR
(*TLBuz Special Warning 3 Behaviour*)
VAR
	p_tTLWarn3BlinkTm : REFERENCE TO TIME;
	p_tBuzWarn3OnTm : REFERENCE TO TIME;
	p_tBuzWarn3RestTm : REFERENCE TO TIME;
	p_usiBuzWarn3OnCntr : REFERENCE TO USINT;
	p_bBuzWarn3StopSeqEn : REFERENCE TO BOOL;
	p_usiBuzWarn3StopSeqCntr : REFERENCE TO USINT;
END_VAR
(*TLBuz Special Warning 4 Behaviour*)
VAR
	p_tTLWarn4BlinkTm : REFERENCE TO TIME;
	p_tBuzWarn4OnTm : REFERENCE TO TIME;
	p_tBuzWarn4RestTm : REFERENCE TO TIME;
	p_usiBuzWarn4OnCntr : REFERENCE TO USINT;
	p_bBuzWarn4StopSeqEn : REFERENCE TO BOOL;
	p_usiBuzWarn4StopSeqCntr : REFERENCE TO USINT;
END_VAR
(*TLBuz Special Warning 5 Behaviour*)
VAR
	p_tTLWarn5BlinkTm : REFERENCE TO TIME;
	p_tBuzWarn5OnTm : REFERENCE TO TIME;
	p_tBuzWarn5RestTm : REFERENCE TO TIME;
	p_usiBuzWarn5OnCntr : REFERENCE TO USINT;
	p_bBuzWarn5StopSeqEn : REFERENCE TO BOOL;
	p_usiBuzWarn5StopSeqCntr : REFERENCE TO USINT;
END_VAR
(*TLBuz Special Buz Behaviour*)
VAR
	p_tBuzAlertOnTm : REFERENCE TO TIME;
	p_tBuzAlertRestTm : REFERENCE TO TIME;
	p_usiBuzAlertOnCntr : REFERENCE TO USINT;
	p_bBuzAlertStopSeqEn : REFERENCE TO BOOL;
	p_usiBuzAlertStopSeqCntr : REFERENCE TO USINT;
END_VAR
(*TLBuz Special Ops TL Behaviour*)
VAR
	p_tTLBlueBlinkTm : REFERENCE TO TIME;
	p_tTLAmberBlinkTm : REFERENCE TO TIME;
	p_tTLWhiteBlinkTm : REFERENCE TO TIME;
	p_tTLRedBlinkTm : REFERENCE TO TIME;
	p_tTLGreenBlinkTm : REFERENCE TO TIME;
END_VAR
(**)
VAR
	p_bCoverSwitchSig : REFERENCE TO BOOL;
	p_eTLBuzMode : REFERENCE TO eTLBuzMod;
	p_bAOIErrSig : REFERENCE TO BOOL;
	p_bAOIOriginSig : REFERENCE TO BOOL;
	p_bBuzAlertEn : REFERENCE TO BOOL;
	p_bTLBlueFlashEn : REFERENCE TO BOOL;
	p_bTLAmberFlashEn : REFERENCE TO BOOL;
	p_bTLWhiteFlashEn : REFERENCE TO BOOL;
	p_bTLRedFlashEn : REFERENCE TO BOOL;
	p_bTLGreenFlashEn : REFERENCE TO BOOL;
END_VAR
(*Add*)
VAR
	p_tyBuffer1BffrStat : REFERENCE TO tyBffrStat;
	p_tyBuffer2BffrStat : REFERENCE TO tyBffrStat;
	p_tyBuffer3BffrStat : REFERENCE TO tyBffrStat;
	p_eMcParamMagExMode : REFERENCE TO eMcMagExchangeMode;
	p_bMcParamAGVComEn : REFERENCE TO BOOL;
END_VAR
```

#### InputRef_Link.var - not listed in the package file held
```iecst
(*2019-04-09*)
VAR
	p_bLinkAlarmWarning : REFERENCE TO BOOL;
	p_bLinkAlarmInfo : REFERENCE TO BOOL;
	p_bLinkUIWarning : REFERENCE TO BOOL;
	p_bLinkAlarmInfoLF : REFERENCE TO BOOL;
	p_bLinkLFBuzMute : REFERENCE TO BOOL;
	p_bLinkAlarmInfoMagFull : REFERENCE TO BOOL;
	p_bLinkMagFullTLMuteBuzz : REFERENCE TO BOOL;
END_VAR
(**)
(*MEK*)
VAR
	p_bLinkAOIOrgOK1 : REFERENCE TO BOOL;
	p_bLinkAOIOrgOK2 : REFERENCE TO BOOL;
	p_bLinkAOIErr1 : REFERENCE TO BOOL;
	p_bLinkAOIErr2 : REFERENCE TO BOOL;
	p_usiLinkMcMod : REFERENCE TO USINT;
END_VAR
(**)
(*BHTC*)
VAR
	p_bLinkMagazineEmpty : REFERENCE TO BOOL;
	p_bLinkUpperMagazineFull : REFERENCE TO BOOL;
	p_bLinkLowerMagazineEmpty : REFERENCE TO BOOL;
	p_bLinkStackEmpty : REFERENCE TO BOOL;
	p_bLinkStackAlmostEmpty : REFERENCE TO BOOL;
	p_bLinkSPIBadPCB : REFERENCE TO BOOL;
	p_bLinkRescanning : REFERENCE TO BOOL;
	p_bLinkRescanFail : REFERENCE TO BOOL;
	p_bLinkBadRejected : REFERENCE TO BOOL;
	p_bLinkBadRejectedwithUBAB : REFERENCE TO BOOL;
	p_bLinkCounterUp : REFERENCE TO BOOL;
	p_bLinkCounterUpNHalf : REFERENCE TO BOOL;
	p_bLinkOvenInfoReceived : REFERENCE TO BOOL;
	p_bLinkThresholdSignal : REFERENCE TO BOOL;
	p_bLinkTwoPCBRejected : REFERENCE TO BOOL;
	p_bLinkUpperMagazineEmpty : REFERENCE TO BOOL;
	p_bLinkLowerMagazineFull : REFERENCE TO BOOL;
END_VAR
(**)
```

#### Act_InitGlobal.st - not listed in the package file held
```iecst
(** 2019-05-20 **)
ACTION Act_InitGlobal:

	//Pass Data To Link
	p_bLinkAlarmWarning ACCESS p_AlarmWarning;
	p_bLinkAlarmInfo ACCESS p_AlarmInfo;
	p_bLinkAlarmInfoLF ACCESS p_AlarmInfoLF;
	p_bLinkLFBuzMute ACCESS p_McParamLFBuzMute;
	p_bLinkAlarmInfoMagFull ACCESS p_OpsMagConvUL1MagFullInfo;
	p_bLinkMagFullTLMuteBuzz ACCESS p_OpsMagConvUL1TLMuteBuzz;

	//Pass Data To Internal Use
	p_bManual ACCESS p_UIUIMnlMod;
	p_bStartup ACCESS p_StartupRun;
	p_bErr ACCESS p_AlarmErr;
	p_bSeqStop ACCESS p_OpsStatusCycleStop;
	p_bStep ACCESS p_OpsStatusStep;
	p_bOps ACCESS p_OpsStatusRun;
	p_bStandby ACCESS p_OpsStatusStop;
	p_bMuteBuz ACCESS p_UIMuteBuz;

	//  -----------------------------------------  TLBuz 5.00.2  -----------------------------------------	//

	p_tTLChgRcpBlinkTm ACCESS p_NtParamTLChgRcpBlinkTm;

	p_tTLErrBlinkTm ACCESS p_NtParamTLErrBlinkTm;
	p_tBuzErrOnTm ACCESS p_NtParamBuzErrOnTm;
	p_tBuzErrRestTm ACCESS p_NtParamBuzErrRestTm;
	p_usiBuzErrOnCntr ACCESS p_NtParamBuzErrOnCntr;
	p_bBuzErrStopSeqEn ACCESS p_NtParamBuzErrStopSeqEn;
	p_usiBuzErrStopSeqCntr ACCESS p_NtParamBuzErrStopSeqCntr;

	p_tTLWarnBlinkTm ACCESS p_NtParamTLWarnBlinkTm;
	p_tBuzWarnOnTm ACCESS p_NtParamBuzWarnOnTm;
	p_tBuzWarnRestTm ACCESS p_NtParamBuzWarnRestTm;
	p_usiBuzWarnOnCntr ACCESS p_NtParamBuzWarnOnCntr;
	p_bBuzWarnStopSeqEn ACCESS p_NtParamBuzWarnStopSeqEn;
	p_usiBuzWarnStopSeqCntr ACCESS p_NtParamBuzWarnStopSeqCntr;

	p_tTLWarn1BlinkTm ACCESS p_NtParamTLWarn1BlinkTm;
	p_tBuzWarn1OnTm ACCESS p_NtParamBuzWarn1OnTm;
	p_tBuzWarn1RestTm ACCESS p_NtParamBuzWarn1RestTm;
	p_usiBuzWarn1OnCntr ACCESS p_NtParamBuzWarn1OnCntr;
	p_bBuzWarn1StopSeqEn ACCESS p_NtParamBuzWarn1StopSeqEn;
	p_usiBuzWarn1StopSeqCntr ACCESS p_NtParamBuzWarn1StopSeqCntr;

	p_tTLWarn2BlinkTm ACCESS p_NtParamTLWarn2BlinkTm;
	p_tBuzWarn2OnTm ACCESS p_NtParamBuzWarn2OnTm;
	p_tBuzWarn2RestTm ACCESS p_NtParamBuzWarn2RestTm;
	p_usiBuzWarn2OnCntr ACCESS p_NtParamBuzWarn2OnCntr;
	p_bBuzWarn2StopSeqEn ACCESS p_NtParamBuzWarn2StopSeqEn;
	p_usiBuzWarn2StopSeqCntr ACCESS p_NtParamBuzWarn2StopSeqCntr;

	p_tTLWarn3BlinkTm ACCESS p_NtParamTLWarn3BlinkTm;
	p_tBuzWarn3OnTm ACCESS p_NtParamBuzWarn3OnTm;
	p_tBuzWarn3RestTm ACCESS p_NtParamBuzWarn3RestTm;
	p_usiBuzWarn3OnCntr ACCESS p_NtParamBuzWarn3OnCntr;
	p_bBuzWarn3StopSeqEn ACCESS p_NtParamBuzWarn3StopSeqEn;
	p_usiBuzWarn3StopSeqCntr ACCESS p_NtParamBuzWarn3StopSeqCntr;

	p_tTLWarn4BlinkTm ACCESS p_NtParamTLWarn4BlinkTm;
	p_tBuzWarn4OnTm ACCESS p_NtParamBuzWarn4OnTm;
	p_tBuzWarn4RestTm ACCESS p_NtParamBuzWarn4RestTm;
	p_usiBuzWarn4OnCntr ACCESS p_NtParamBuzWarn4OnCntr;
	p_bBuzWarn4StopSeqEn ACCESS p_NtParamBuzWarn4StopSeqEn;
	p_usiBuzWarn4StopSeqCntr ACCESS p_NtParamBuzWarn4StopSeqCntr;

	p_tTLWarn5BlinkTm ACCESS p_NtParamTLWarn5BlinkTm;
	p_tBuzWarn5OnTm ACCESS p_NtParamBuzWarn5OnTm;
	p_tBuzWarn5RestTm ACCESS p_NtParamBuzWarn5RestTm;
	p_usiBuzWarn5OnCntr ACCESS p_NtParamBuzWarn5OnCntr;
	p_bBuzWarn5StopSeqEn ACCESS p_NtParamBuzWarn5StopSeqEn;
	p_usiBuzWarn5StopSeqCntr ACCESS p_NtParamBuzWarn5StopSeqCntr;

	p_tBuzAlertOnTm ACCESS p_NtParamBuzAlertOnTm;
	p_tBuzAlertRestTm ACCESS p_NtParamBuzAlertRestTm;
	p_usiBuzAlertOnCntr ACCESS p_NtParamBuzAlertOnCntr;
	p_bBuzAlertStopSeqEn ACCESS p_NtParamBuzAlertStopSeqEn;
	p_usiBuzAlertStopSeqCntr ACCESS p_NtParamBuzAlertStopSeqCntr;

	p_tTLBlueBlinkTm ACCESS p_NtParamTLBlueBlinkTm;
	p_tTLAmberBlinkTm ACCESS p_NtParamTLAmberBlinkTm;
	p_tTLWhiteBlinkTm ACCESS p_NtParamTLWhiteBlinkTm;
	p_tTLRedBlinkTm ACCESS p_NtParamTLRedBlinkTm;
	p_tTLGreenBlinkTm ACCESS p_NtParamTLGreenBlinkTm;

	//  ----------------------------------------------  ||  ---------------------------------------------	//

	p_bCoverSwitchSig ACCESS p_DICoverSWSig;
	p_eTLBuzMode ACCESS p_NtParamTLBuzMode;

	p_bMcParamAGVComEn ACCESS p_McParamAGVComEn; //Add
	p_eMcParamMagExMode ACCESS p_McParamMagExMode;

	p_tyBuffer1BffrStat ACCESS p_Buffer1BffrStat; //ADD
	p_tyBuffer2BffrStat ACCESS p_Buffer2BffrStat; //ADD
	p_tyBuffer3BffrStat ACCESS p_Buffer3BffrStat; //ADD
	(* Always Change If Project Change *)

END_ACTION
```

#### Act_InitLocal.st - not listed in the package file held
```iecst
(** 2020-03-16 **)
ACTION Act_InitLocal:

	//Input Reference Link To Local Variable
	p_eAct ACCESS ADR(eAct);
	p_bManual ACCESS ADR(bManual);
	p_bStartup ACCESS ADR(bStartup);
	p_bErr ACCESS ADR(bErr);
	p_bErrNoBuz ACCESS ADR(bErrNoBuz);
	p_bWarning ACCESS ADR(bWarning);
	p_bWarningNoBuz ACCESS ADR(bWarningNoBuz);
	p_bWarning1 ACCESS ADR(bWarning1);
	p_bWarning1NoBuz ACCESS ADR(bWarning1NoBuz);
	p_bWarning2 ACCESS ADR(bWarning2);
	p_bWarning2NoBuz ACCESS ADR(bWarning2NoBuz);
	p_bWarning3 ACCESS ADR(bWarning3);
	p_bWarning3NoBuz ACCESS ADR(bWarning3NoBuz);
	p_bWarning4 ACCESS ADR(bWarning4);
	p_bWarning4NoBuz ACCESS ADR(bWarning4NoBuz);
	p_bWarning5 ACCESS ADR(bWarning5);
	p_bWarning5NoBuz ACCESS ADR(bWarning5NoBuz);
	p_bChgRcp ACCESS ADR(bChgRcp);
	p_bSeqStop ACCESS ADR(bSeqStop);
	p_bStep ACCESS ADR(bStep);
	p_bOps ACCESS ADR(bOps);
	p_bStandby ACCESS ADR(bStandby);
	p_bSimulation ACCESS ADR(bSimulation);
	p_bMuteBuz ACCESS ADR(bMuteBuz);

	p_tTLChgRcpBlinkTm ACCESS ADR(tTLChgRcpBlinkTm);

	p_tTLErrBlinkTm ACCESS ADR(tTLErrBlinkTm);
	p_tBuzErrOnTm ACCESS ADR(tBuzErrOnTm);
	p_tBuzErrRestTm ACCESS ADR(tBuzErrRestTm);
	p_usiBuzErrOnCntr ACCESS ADR(usiBuzErrOnCntr);
	p_bBuzErrStopSeqEn ACCESS ADR(bBuzErrStopSeqEn);
	p_usiBuzErrStopSeqCntr ACCESS ADR(usiBuzErrStopSeqCntr);

	p_tTLWarnBlinkTm ACCESS ADR(tTLWarnBlinkTm);
	p_tBuzWarnOnTm ACCESS ADR(tBuzWarnOnTm);
	p_tBuzWarnRestTm ACCESS ADR(tBuzWarnRestTm);
	p_usiBuzWarnOnCntr ACCESS ADR(usiBuzWarnOnCntr);
	p_bBuzWarnStopSeqEn ACCESS ADR(bBuzWarnStopSeqEn);
	p_usiBuzWarnStopSeqCntr ACCESS ADR(usiBuzWarnStopSeqCntr);

	p_tTLWarn1BlinkTm ACCESS ADR(tTLWarn1BlinkTm);
	p_tBuzWarn1OnTm ACCESS ADR(tBuzWarn1OnTm);
	p_tBuzWarn1RestTm ACCESS ADR(tBuzWarn1RestTm);
	p_usiBuzWarn1OnCntr ACCESS ADR(usiBuzWarn1OnCntr);
	p_bBuzWarn1StopSeqEn ACCESS ADR(bBuzWarn1StopSeqEn);
	p_usiBuzWarn1StopSeqCntr ACCESS ADR(usiBuzWarn1StopSeqCntr);

	p_tTLWarn2BlinkTm ACCESS ADR(tTLWarn2BlinkTm);
	p_tBuzWarn2OnTm ACCESS ADR(tBuzWarn2OnTm);
	p_tBuzWarn2RestTm ACCESS ADR(tBuzWarn2RestTm);
	p_usiBuzWarn2OnCntr ACCESS ADR(usiBuzWarn2OnCntr);
	p_bBuzWarn2StopSeqEn ACCESS ADR(bBuzWarn2StopSeqEn);
	p_usiBuzWarn2StopSeqCntr ACCESS ADR(usiBuzWarn2StopSeqCntr);

	p_tTLWarn3BlinkTm ACCESS ADR(tTLWarn3BlinkTm);
	p_tBuzWarn3OnTm ACCESS ADR(tBuzWarn3OnTm);
	p_tBuzWarn3RestTm ACCESS ADR(tBuzWarn3RestTm);
	p_usiBuzWarn3OnCntr ACCESS ADR(usiBuzWarn3OnCntr);
	p_bBuzWarn3StopSeqEn ACCESS ADR(bBuzWarn3StopSeqEn);
	p_usiBuzWarn3StopSeqCntr ACCESS ADR(usiBuzWarn3StopSeqCntr);

	p_tTLWarn4BlinkTm ACCESS ADR(tTLWarn4BlinkTm);
	p_tBuzWarn4OnTm ACCESS ADR(tBuzWarn4OnTm);
	p_tBuzWarn4RestTm ACCESS ADR(tBuzWarn4RestTm);
	p_usiBuzWarnOnCntr ACCESS ADR(usiBuzWarn4OnCntr);
	p_bBuzWarn4StopSeqEn ACCESS ADR(bBuzWarn4StopSeqEn);
	p_usiBuzWarn4StopSeqCntr ACCESS ADR(usiBuzWarn4StopSeqCntr);

	p_tTLWarn5BlinkTm ACCESS ADR(tTLWarn5BlinkTm);
	p_tBuzWarn5OnTm ACCESS ADR(tBuzWarn5OnTm);
	p_tBuzWarn5RestTm ACCESS ADR(tBuzWarn5RestTm);
	p_usiBuzWarn5OnCntr ACCESS ADR(usiBuzWarn5OnCntr);
	p_bBuzWarn5StopSeqEn ACCESS ADR(bBuzWarn5StopSeqEn);
	p_usiBuzWarn5StopSeqCntr ACCESS ADR(usiBuzWarn5StopSeqCntr);

	p_tBuzAlertOnTm ACCESS ADR(tBuzAlertOnTm);
	p_tBuzAlertRestTm ACCESS ADR(tBuzAlertRestTm);
	p_usiBuzAlertOnCntr ACCESS ADR(usiBuzAlertOnCntr);
	p_bBuzAlertStopSeqEn ACCESS ADR(bBuzAlertStopSeqEn);
	p_usiBuzAlertStopSeqCntr ACCESS ADR(usiBuzAlertStopSeqCntr);

	p_tTLBlueBlinkTm ACCESS ADR(tTLBlueBlinkTm);
	p_tTLAmberBlinkTm ACCESS ADR(tTLAmberBlinkTm);
	p_tTLWhiteBlinkTm ACCESS ADR(tTLWhiteBlinkTm);
	p_tTLRedBlinkTm ACCESS ADR(tTLRedBlinkTm);
	p_tTLGreenBlinkTm ACCESS ADR(tTLGreenBlinkTm);

	p_bCoverSwitchSig ACCESS ADR(bCoveSwitchSig);
	p_eTLBuzMode ACCESS ADR(eTLBuzMode);
	p_bAOIErrSig ACCESS ADR(bAOIErrSig);
	p_bAOIOriginSig ACCESS ADR(bAOIOriginSig);

	p_bBuzAlertEn ACCESS ADR(bBuzAlertEn);
	p_bTLBlueFlashEn ACCESS ADR(bTLBlueFlashEn);
	p_bTLAmberFlashEn ACCESS ADR(bTLAmberFlashEn);
	p_bTLWhiteFlashEn ACCESS ADR(bTLWhiteFlashEn);
	p_bTLRedFlashEn ACCESS ADR(bTLRedFlashEn);
	p_bTLGreenFlashEn ACCESS ADR(bTLGreenFlashEn);

END_ACTION
```

#### Act_Link.st - not listed in the package file held
```iecst
(** 2019-03-29 **)
ACTION Act_Link:

	p_bWarning			:= p_bLinkAlarmWarning OR (p_bLinkAlarmInfo AND NOT (p_bLinkAlarmInfoLF AND p_bLinkLFBuzMute) AND NOT(p_bLinkAlarmInfoMagFull AND p_bLinkMagFullTLMuteBuzz));

	p_bWarningNoBuz		:= (p_bLinkAlarmInfoLF AND p_bLinkLFBuzMute) OR (p_bLinkAlarmInfoMagFull AND p_bLinkMagFullTLMuteBuzz);

END_ACTION
```

### Alarm.typ - Do Not Change!!!
```iecst
(*2019-03-25*)
(**)

TYPE
	eAlarmAction :
		(
		AlarmActIdle,
		AlarmActCreateDir,
		AlarmActDeleteOldLog,
		AlarmActReadHistory,
		AlarmActWriteHistory,
		AlarmActAppendLog,
		AlarmActAppendLogWriteHistory,
		AlarmActResetHistory,
		AlarmActBGStartLog,
		AlarmActBGStopLog
		);
END_TYPE

(**)

TYPE
	tyAlarmCurr : 	STRUCT
		eSeverity : eAlmSeverity;
		sMsg : STRING[300];
		bAlm : BOOL;
		bWarning : BOOL;
		udiErrorCode : UDINT;
		sProgNm : STRING[15];
		sDT : STRING[80];
		udiModErrCode : UDINT;
	END_STRUCT;
	tyHistory : 	STRUCT
		sDT : STRING[80];
		sProgNm : STRING[15];
		udiModErrCode : UDINT;
		udiErrorCode : UDINT;
	END_STRUCT;
	tyAlmProgNm : 	STRUCT
		sAWOpenProgNm : STRING[15];
		sAWCloseProgNm : STRING[15];
		sMagAWOpenProgNm : STRING[15];
		sTravProgNm : STRING[15];
		sLifterBtmProgNm : STRING[15];
		sConvProgNm : STRING[15];
		sDCConvProgNm : STRING[15];
		sMagConvProgNm : STRING[15];
		sMagConv2ClpProgNm : STRING[15];
		sBufferProgNm : STRING[15];
		sMotorBrkProgNm : STRING[15];
		sMtrPshrProgNm : STRING[15];
		sStepperProgNm : STRING[15];
		sPneuNoSenProgNm : STRING[15];
		sPneuExtSenProgNm : STRING[15];
		sPneuRetSenProgNm : STRING[15];
		sPneu2SenProgNm : STRING[15];
		sPneu3SenProgNm : STRING[15];
		sUSSMEMAProgNm : STRING[15];
		sDSSMEMAProgNm : STRING[15];
		sHermesProgNm : STRING[15];
		sUSHermesAProgNm : STRING[15];
		sUSHermesBProgNm : STRING[15];
		sDSHermesProgNm : STRING[15];
		sRmtHermesProgNm : STRING[15];
		sLFLeaderProgNm : STRING[15];
		sLFFollowerProgNm : STRING[15];
		sLCSProgNm : STRING[15];
		sLCSLFProgNm : STRING[15];
		sLCSMngRcpProgNm : STRING[15];
		sTCPProgNm : STRING[15];
		sUSSOTProgNm : STRING[15];
		sDSSOTProgNm : STRING[15];
		sBarcodeRdrProgNm : STRING[15];
		sRS232MirtecProgNm : STRING[15];
		sProdRcpProgNm : STRING[15];
		sMagRcpProgNm : STRING[15];
		sMpProdRcpProgNm : STRING[15];
		sAlarmProgNm : STRING[15];
		sNtParamProgNm : STRING[15];
		sMcParamProgNm : STRING[15];
		sUsrMgmtProgNm : STRING[15];
		sLibVerProgNm : STRING[15];
		sUsrFolderProgNm : STRING[15];
		sHWInfoProgNm : STRING[15];
		sDInputProgNm : STRING[15];
		sTimeProgNm : STRING[15];
		sMachineProgNm : STRING[15];
		sOps1ProgNm : STRING[15];
		sOpsTravLifULProgNm : STRING[15];
		sOpsMagConvULProgNm : STRING[15];
		sOpsMagConvUL2ProgNm : STRING[15];
		sOpsMagConvUL3ProgNm : STRING[15];
		sOpsLifMagULProgNm : STRING[15];
		sOpsInMagConvProgNm : STRING[15];
		sOpsOutMagConvProgNm : STRING[15];
		sOpsMagConvStprProgNm : STRING[15];
		sOpsMagConvStpr2ProgNm : STRING[15];
		sWarningLibVersion : STRING[15];
		sAGVComProgNm : STRING[15];
		sAGVProgNm : STRING[15];
		sFrameProgNm : STRING[15];
		sLiberWarnName : STRING[15];
		sSimu1ProgNm : STRING[15];
		sSvyHermesProgNm : STRING[15];
		sAutoRcpProgNm : STRING[15];
	END_STRUCT;
	tyAlmIn1 : 	STRUCT
		udiRstErr : UDINT;
		eAct : eAlarmAction;
		dtCurrDT : DATE_AND_TIME;
		udiFileKeepDay : UDINT;
		sProgNm : STRING[15];
		bStartupUISettingsLoadDone : BOOL;
	END_STRUCT;
	tyAlmOut1 : 	STRUCT
		bWarning : BOOL;
		bInfo : BOOL;
		bErr : BOOL;
		bInfoLF : BOOL;
		eStat : eAlarmAction;
		eStatus : eFBStatus;
		a_tyCurrList : ARRAY[1..c_udiAlarmCurrMax]OF tyAlarmCurr;
		a_udiRecoveryList : ARRAY[1..c_udiAlarmCurrMax]OF UDINT;
		sInfoMsg : STRING[100];
		sStatTxt : STRING[200];
		bHistoryFileNotFound : BOOL;
	END_STRUCT;
	tyAlarm : 	STRUCT
		In : tyAlmIn1;
		Out : tyAlmOut1;
	END_STRUCT;
END_TYPE
```

### Alarm.var - Change By Project
```iecst
(*2019-03-25*)
VAR
	g_tyAlmProgNm : tyAlmProgNm;
	g_tyAlm : tyAlmOut1;
END_VAR
(**)
(*Constant*)
VAR CONSTANT
	c_udiAlarmCurrMax : UDINT := 200;
	c_udiAlarmHistoryMax : UDINT := 300;
END_VAR
(**)
```

### Program Logical/Alarm/Alarm (IEC, version 1.00.0) - 1.00.0 - NtLogFile v5.00.0 , NtFileIO v5.00.0

#### Init.st - Change By Project
```iecst
(** 2019-03-25 **)
PROGRAM _INIT

	(* Always Change If Project Change *)

	//Pass Address To Global Address For External Use
	//Action, State & Status
	p_AlarmStat		:= ADR(eStat);
	p_AlarmStatus	:= ADR(eStatus);
	p_AlarmStatTxt	:= ADR(sStatTxt);

	//Alarm

	//Output
	p_AlarmErr					:= ADR(bErr);
	p_AlarmWarning				:= ADR(bWarning);
	p_AlarmCurrList				:= ADR(a_tyCurrList);
	p_AlarmRecoveryList			:= ADR(a_udiRecoveryList);
	p_AlarmHistoryList			:= ADR(a_sHistoryList);
	p_AlarmInfo					:= ADR(bInfo);
	p_AlarmInfoLF				:= ADR(bInfoLF);
	p_AlarmInfoMsg				:= ADR(sInfoMsg);
	p_AlarmHistoryFileNotFound	:= ADR(bHistoryFileNotFound);

	(* Always Change If Project Change *)

END_PROGRAM
```

#### Act_InitGlobal.st - Change By Project
```iecst
(** 2019-03-25 **)
ACTION Act_InitGlobal:

	(* Always Change If Project Change *)

	//Pass Data To Link
	p_tyLinkUsrFolderAlmData ACCESS p_UsrFolderAlmData;
	p_tyLinkLibVerAlmData ACCESS p_LibVerAlmData;
	p_tyLinkTimeAlmData ACCESS p_TimeAlmData;
	p_tyLinkTimeAlmData1 ACCESS p_TimeAlmData1;
	p_tyLinkHWInfoAlmData ACCESS p_HWInfoAlmData;
	p_tyLinkProdRcpAlmData ACCESS p_ProdRcpAlmData;
	p_tyLinkMpProdRcpAlmData ACCESS p_MpProdRcpAlmData;
	p_tyLinkMagRcpAlmData ACCESS p_MagRcpAlmData;
	p_tyLinkMcParamAlmData ACCESS p_McParamAlmData;
	p_tyLinkNtParamAlmData ACCESS p_NtParamAlmData;
	p_tyLinkUsrMgmtAlmData ACCESS p_UsrMgmtAlmData;
	p_tyLinkBuffer1AlmData ACCESS p_Buffer1AlmData;
	p_tyLinkBuffer2AlmData ACCESS p_Buffer2AlmData;
	p_tyLinkBuffer3AlmData ACCESS p_Buffer3AlmData;
	p_tyLinkUSSMEMAAAlmData ACCESS p_USSMEMAAAlmData;
	p_tyLinkUSSMEMABAlmData ACCESS p_USSMEMABAlmData;
	p_tyLinkUSSMEMA1AlmData ACCESS p_USSMEMA1AlmData;
	p_tyLinkUSSMEMA2AlmData ACCESS p_USSMEMA2AlmData;
	p_tyLinkUSSMEMA3AlmData ACCESS p_USSMEMA3AlmData;
	p_tyLinkDSSMEMA1AlmData ACCESS p_DSSMEMA1AlmData;
	p_tyLinkDSSMEMA2AlmData ACCESS p_DSSMEMA2AlmData;
	p_tyLinkDSSMEMA3AlmData ACCESS p_DSSMEMA3AlmData;
	p_tyLinkInShutterAlmData ACCESS p_Pneu2SenInShutterAlmData;
	p_tyLinkOutShutterAlmData ACCESS p_Pneu2SenOutShutterAlmData;
	p_tyLinkOutShutterAlmData2 ACCESS p_Pneu2SenOutShutterAlmData2;
	p_tyLinkOutShutterAlmData3 ACCESS p_Pneu2SenOutShutterAlmData3;
	p_tyLinkStopperAAlmData ACCESS p_PneuNoSenStopperAAlmData;
	p_tyLinkStopperBAlmData ACCESS p_PneuNoSenStopperBAlmData;
	p_tyLinkPshrConvAlmData ACCESS p_PshrConvAlmData;
	p_tyLinkMagConv1AlmData ACCESS p_MagConv2Clp1AlmData;
	p_tyLinkMagConv2AlmData ACCESS p_MagConv2Clp2AlmData;
	p_tyLinkMagConv3AlmData ACCESS p_MagConv2Clp3AlmData;
	p_tyLinkAWOpenAlmData ACCESS p_AWOpenAlmData;
	p_tyLinkAWOpenAlmData1 ACCESS p_AWOpenAlmData1;
	p_tyLinkAWOpenAlmData2 ACCESS p_AWOpenAlmData2;
	p_tyLinkAWOpenAlmData3 ACCESS p_AWOpenAlmData3;
	p_tyLinkTravAlmData ACCESS p_TravAlmData;
	p_tyLinkTravAlmData1 ACCESS p_TravAlmData1;
	p_tyLinkTravAlmData2 ACCESS p_TravAlmData2;
	p_tyLinkTravAlmData3 ACCESS p_TravAlmData3;
	p_tyLinkLifterBtmAlmData ACCESS p_LifterBtmAlmData;
	p_tyLinkLifterBtmAlmData1 ACCESS p_LifterBtmAlmData1;
	p_tyLinkLifterBtmAlmData2 ACCESS p_LifterBtmAlmData2;
	p_tyLinkLifterBtmAlmData3 ACCESS p_LifterBtmAlmData3;
	p_tyLinkDIAlmData1 ACCESS p_DIAlmData1;
	p_tyLinkDIAlmData2 ACCESS p_DIAlmData2;
	p_tyLinkDIAlmData3 ACCESS p_DIAlmData3;
	p_tyLinkDIAlmData4 ACCESS p_DIAlmData4;
	p_tyLinkDIAlmData5 ACCESS p_DIAlmData5;
	p_tyLinkDIAlmData6 ACCESS p_DIAlmData6;
	p_tyLinkAGVMag1AlmData ACCESS p_AGVMag1AlmData;
	p_tyLinkAGVMag2AlmData ACCESS p_AGVMag2AlmData;
	p_tyLinkAGVMag3AlmData ACCESS p_AGVMag3AlmData;
	p_tyLinkHermesAlmData ACCESS p_HermesAlmData;
	p_tyLinkUSHermesAAlmData ACCESS p_USHermesAAlmData;
	p_tyLinkUSHermesAAlmData1 ACCESS p_USHermesAAlmData1;
	p_tyLinkUSHermesAAlmData2 ACCESS p_USHermesAAlmData2;
	p_tyLinkUSHermesAAlmData3 ACCESS p_USHermesAAlmData3;
	p_tyLinkUSHermesAAlmData4 ACCESS p_USHermesAAlmData4;
	p_tyLinkUSHermesAAlmData5 ACCESS p_USHermesAAlmData5;
	p_tyLinkUSHermesAInfoData ACCESS p_USHermesAInfoData;
	p_tyLinkUSHermesBAlmData ACCESS p_USHermesBAlmData;
	p_tyLinkUSHermesBAlmData1 ACCESS p_USHermesBAlmData1;
	p_tyLinkUSHermesBAlmData2 ACCESS p_USHermesBAlmData2;
	p_tyLinkUSHermesBAlmData3 ACCESS p_USHermesBAlmData3;
	p_tyLinkUSHermesBAlmData4 ACCESS p_USHermesBAlmData4;
	p_tyLinkUSHermesBAlmData5 ACCESS p_USHermesBAlmData5;
	p_tyLinkUSHermesBInfoData ACCESS p_USHermesBInfoData;
	p_tyLinkRmtHermesAlmData ACCESS p_RmtHermesAlmData;
	p_tyLinkRmtHermesAlmData1 ACCESS p_RmtHermesAlmData1;
	p_tyLinkRmtHermesAlmData2 ACCESS p_RmtHermesAlmData2;
	p_tyLinkRmtHermesAlmData3 ACCESS p_RmtHermesAlmData3;
	//Svy Hermes
	p_tyLinkSvyHermesAlmData ACCESS p_SvyHermesAlmData;
	p_tyLinkSvyHermesAlmData1 ACCESS p_SvyHermesAlmData1;
	p_tyLinkSvyHermesAlmData2 ACCESS p_SvyHermesAlmData2;
	p_tyLinkSvyHermesAlmData3 ACCESS p_SvyHermesAlmData3;
	p_tyLinkSvyHermesAlmData4 ACCESS p_SvyHermesAlmData4;
	p_tyLinkSvyHermesInfoData ACCESS p_SvyHermesInfoData;
	p_tyLinkSvyHermesInfoData1 ACCESS p_SvyHermesInfoData1;
	p_tyLinkSvyHermesInfoData2 ACCESS p_SvyHermesInfoData2;
	p_tyLinkSvyHermesInfoData3 ACCESS p_SvyHermesInfoData3;
	p_tyLinkSvyHermesInfoData4 ACCESS p_SvyHermesInfoData4;

	p_tyLinkLFLeaderAlmData ACCESS p_LFLeaderAlmData;
	p_tyLinkLFFollowerAlmData ACCESS p_LFFollowerAlmData;
	p_tyLinkLFFollowerInfoData ACCESS p_LFFollowerInfoData;
	p_tyLinkLFFollowerInfoData1 ACCESS p_LFFollowerInfoData1;
	p_tyLinkFollower1AlmData ACCESS p_Follower1AlmData;
	p_tyLinkFollower1InfoData ACCESS p_Follower1InfoData;
	p_tyLinkFollower1InfoData1 ACCESS p_Follower1InfoData1;
	p_tyLinkFollower2AlmData ACCESS p_Follower2AlmData;
	p_tyLinkFollower2InfoData ACCESS p_Follower2InfoData;
	p_tyLinkFollower2InfoData1 ACCESS p_Follower2InfoData1;
	p_tyLinkLCSMngRcpAlmData ACCESS p_LCSMngRcpAlmData;
	p_tyLinkLCSLFAlmData ACCESS p_LCSLFAlmData;
	p_tyLinkLCSLFInfoData ACCESS p_LCSLFInfoData;
	p_tyLinkOpsTravLifULAlmData ACCESS p_OpsTravLifULAlmData;
//	p_tyLinkOpsMagUL1AlmData ACCESS p_OpsMagUL1AlmData;
//	p_tyLinkOpsMagUL1AlmData1 ACCESS p_OpsMagUL1AlmData1;
//	p_tyLinkOpsMagUL2AlmData ACCESS p_OpsMagUL2AlmData;
//	p_tyLinkOpsMagUL2AlmData1 ACCESS p_OpsMagUL2AlmData1;
//	p_tyLinkOpsMagUL3AlmData ACCESS p_OpsMagUL3AlmData;
//	p_tyLinkOpsMagUL3AlmData1 ACCESS p_OpsMagUL3AlmData1;
	p_tyLinkOpsLifMagULAlmData ACCESS p_OpsLifMagULAlmData;
	p_tyLinkOpsLifMagULAlmData1 ACCESS p_OpsLifMagULAlmData1;
	p_tyLinkOpsLifMagULAlmData2 ACCESS p_OpsLifMagULAlmData2;

	p_tyLinkOpsMagConvUL1AlmData ACCESS p_OpsMagConvUL1AlmData;
	p_tyLinkOpsMagConvUL1AlmData1 ACCESS p_OpsMagConvUL1AlmData1;
	p_tyLinkOpsMagConvUL2AlmData ACCESS p_OpsMagConvUL2AlmData;
	p_tyLinkOpsMagConvUL2AlmData1 ACCESS p_OpsMagConvUL2AlmData1;
	p_tyLinkOpsMagConvUL3AlmData ACCESS p_OpsMagConvUL3AlmData;
	p_tyLinkOpsMagConvUL3AlmData1 ACCESS p_OpsMagConvUL3AlmData1;
	p_tyLinkMag1SafetyBarAlmData ACCESS p_Pneu2SMag1SafetyBarAlmData;
	p_tyLinkMag2SafetyBarAlmData ACCESS p_Pneu2SMag2SafetyBarAlmData;
	p_tyLinkMag3SafetyBarAlmData ACCESS p_Pneu2SMag3SafetyBarAlmData;
	p_tyLinkMag1AWEngageAlmData ACCESS p_Pneu2SMag1AWEngageAlmData;
	p_tyLinkMag2AWEngageAlmData ACCESS p_Pneu2SMag2AWEngageAlmData;
	p_tyLinkMag3AWEngageAlmData ACCESS p_Pneu2SMag3AWEngageAlmData;
	p_tyLinkMagAWOpen1AlmData ACCESS p_MagAWOpen1AlmData;
	p_tyLinkMagAWOpen1AlmData1 ACCESS p_MagAWOpen1AlmData1;
	p_tyLinkMagAWOpen1AlmData2 ACCESS p_MagAWOpen1AlmData2;
	p_tyLinkMagAWOpen1AlmData3 ACCESS p_MagAWOpen1AlmData3;
	p_tyLinkMagAWOpen2AlmData ACCESS p_MagAWOpen2AlmData;
	p_tyLinkMagAWOpen2AlmData1 ACCESS p_MagAWOpen2AlmData1;
	p_tyLinkMagAWOpen2AlmData2 ACCESS p_MagAWOpen2AlmData2;
	p_tyLinkMagAWOpen2AlmData3 ACCESS p_MagAWOpen2AlmData3;
	p_tyLinkMagAWOpen3AlmData ACCESS p_MagAWOpen3AlmData;
	p_tyLinkMagAWOpen3AlmData1 ACCESS p_MagAWOpen3AlmData1;
	p_tyLinkMagAWOpen3AlmData2 ACCESS p_MagAWOpen3AlmData2;
	p_tyLinkMagAWOpen3AlmData3 ACCESS p_MagAWOpen3AlmData3;
	p_tyLinkMcAlarmData ACCESS p_McAlmData;
	p_tyLinkUSSOT1AlmData ACCESS p_USSOT1AlmData;
	p_tyLinkUSSOT2AlmData ACCESS p_USSOT2AlmData;
	p_tyLinkUSSOT3AlmData ACCESS p_USSOT3AlmData;
	p_tyLinkDSSOT1AlmData ACCESS p_DSSOT1AlmData;
	p_tyLinkDSSOT2AlmData ACCESS p_DSSOT2AlmData;
	p_tyLinkDSSOT3AlmData ACCESS p_DSSOT3AlmData;
	p_tyLinkMag1SelClampAlmData ACCESS p_PneuNoSenSelClamp1AlmData;
	p_tyLinkMag2SelClampAlmData ACCESS p_PneuNoSenSelClamp2AlmData;
	p_tyLinkMag3SelClampAlmData ACCESS p_PneuNoSenSelClamp3AlmData;
	p_tyLinkAGVAlmData1 ACCESS p_AGVAlmData1;
	p_tyLinkAWPushOrPullerAlmData ACCESS p_AWPushOrPullerAlmData;
	p_tyLinkAWPushOrPullerAlmData1 ACCESS p_AWPushOrPullerAlmData1;
	p_tyLinkAWPushOrPullerAlmData2 ACCESS p_AWPushOrPullerAlmData2;
	p_tyLinkAWPushOrPullerAlmData3 ACCESS p_AWPushOrPullerAlmData3;
	p_tyLinkMtrPshrAlmData ACCESS p_MtrPshrAlmData;

	//MagConv Alarm
	p_tyLinkTopEntStprAlmData ACCESS p_PneuNoSenTopEntStprAlmData;
	p_tyLinkTopMidStprAlmData ACCESS p_PneuNoSenTopMidStprAlmData;
	p_tyLinkTopExtStprAlmData ACCESS p_PneuNoSenTopExtStprAlmData;
	p_tyLinkBtmMidStprAlmData ACCESS p_PneuNoSenBtmMidStprAlmData;
	p_tyLinkBtmExtStprAlmData ACCESS p_PneuNoSenBtmExtStprAlmData;
	p_tyLinkTopEntStpr2AlmData ACCESS p_PneuNoSenTopEntStpr2AlmData;
	p_tyLinkTopMidStpr2AlmData ACCESS p_PneuNoSenTopMidStpr2AlmData;
	p_tyLinkTopExtStpr2AlmData ACCESS p_PneuNoSenTopExtStpr2AlmData;
	p_tyLinkBtmMidStpr2AlmData ACCESS p_PneuNoSenBtmMidStpr2AlmData;
	p_tyLinkBtmExtStpr2AlmData ACCESS p_PneuNoSenBtmExtStpr2AlmData;

	p_tyLinkInMagConvAlmData ACCESS p_InMagConvAlmData;
	p_tyLinkOutMagConvAlmData ACCESS p_OutMagConvAlmData;
	p_tyLinkInMagConv2AlmData ACCESS p_InMagConv2AlmData;
	p_tyLinkOutMagConv2AlmData ACCESS p_OutMagConv2AlmData;
	p_tyLinkLifterMagConvAlmData ACCESS p_LifterMagConvAlmData;
	p_tyLinkLifterMagConv2AlmData ACCESS p_LifterMagConv2AlmData;

	p_bNtParamProjMagConvLane1Prep ACCESS p_NtParamProjMagConvLane1Prep;
	p_bNtParamProjMagConvLane2Prep ACCESS p_NtParamProjMagConvLane2Prep;
	p_tyLinkOpsInMagConvAlmData ACCESS p_OpsInMagConvAlmData;
	p_tyLinkOpsOutMagConvAlmData ACCESS p_OpsOutMagConvAlmData;

	p_bNtParamProjLifter2Prep ACCESS p_NtParamProjLifter2Prep;
	p_tyLinkLifter2AlmData ACCESS p_Lifter2AlmData;
	p_tyLinkLifter2AlmData1 ACCESS p_Lifter2AlmData1;
	p_tyLinkLifter2AlmData2 ACCESS p_Lifter2AlmData2;
	p_tyLinkLifter2AlmData3 ACCESS p_Lifter2AlmData3;
	//	p_tyLinkOpsStprAlmData ACCESS p_OpsStprAlmData;
	p_tyLinkPPAlmData ACCESS p_PPAlmData;
	p_tyLinkPPAlmData1 ACCESS p_PPAlmData1;
	p_tyLinkPPAlmData2 ACCESS p_PPAlmData2;
	p_tyLinkPPAlmData3 ACCESS p_PPAlmData3;

	p_bNTParamTCPAGVSigPrep ACCESS p_NtParamProjTCPAGVSigPrep;
	p_tyLinkTCPAlmData ACCESS p_TCPAlmData;
	p_tyLinkTCPAlmData ACCESS p_TCPAlmData; //TCPAGV
	p_tyLinkTCPAlmData1 ACCESS p_TCPAlmData1;
	p_tyLinkTCPAlmData2 ACCESS p_TCPAlmData2;
	p_tyLinkTCPAlmData3 ACCESS p_TCPAlmData3;

	p_bNtParamTCPScannerPrep ACCESS  p_NtParamProjScanPrep;
	p_tyLinkTCPTopAlmData ACCESS p_TCPTopAlmData; //TCPScanner
	p_tyLinkTCPBtmAlmData ACCESS p_TCPBtmAlmData;

	//Auto Rcp
	p_bNtParamAutoRcpPrep ACCESS p_NtParamAutoRcpPrep;
	p_tyLinkAutoRcpAlmData ACCESS  p_AutoRcpAlmData;

	//Pass Data To Internal Use
	p_udiRstErr ACCESS p_RstErrReset;
	p_eAct ACCESS p_StartupAlarmAct;
	p_dtCurrDT ACCESS p_TimeCurrDT;
	p_udiFileKeepDay ACCESS p_NtParamAlmFileKeepDay;
	p_sProgNm ACCESS p_NtParamAlmProgNm;
	p_bNtSettingsLoadDone ACCESS p_StartupNtSettingsLoadDone;
	p_bStartupUISettingsLoadDone ACCESS p_StartupUISettingsLoadDone;
	// ADD

	(* Always Change If Project Change *)

END_ACTION
```

#### InputRef_Link.var - Change By Project
```iecst
(*2019-01-07*)
(*Avoid access (*void) memory*)
VAR
	p_bNtParamProjLifter2Prep : REFERENCE TO BOOL;
	p_bNTParamTCPAGVSigPrep : REFERENCE TO BOOL;
	p_bNtParamTCPScannerPrep : REFERENCE TO BOOL;
	p_bNtParamAutoRcpPrep : REFERENCE TO BOOL;
	p_bNtParamProjMagConvLane1Prep : REFERENCE TO BOOL;
	p_bNtParamProjMagConvLane2Prep : REFERENCE TO BOOL;
END_VAR
(**)
(*External Data*)
VAR
	p_tyLinkUsrFolderAlmData : REFERENCE TO tyAlmDat;
	p_tyLinkLibVerAlmData : REFERENCE TO tyAlmDat;
	p_tyLinkTimeAlmData : REFERENCE TO tyAlmDat;
	p_tyLinkTimeAlmData1 : REFERENCE TO tyAlmDat;
	p_tyLinkHWInfoAlmData : REFERENCE TO tyAlmDat;
	p_tyLinkProdRcpAlmData : REFERENCE TO tyAlmDat;
	p_tyLinkMpProdRcpAlmData : REFERENCE TO tyAlmDat;
	p_tyLinkMagRcpAlmData : REFERENCE TO tyAlmDat;
	p_tyLinkMcParamAlmData : REFERENCE TO tyAlmDat;
	p_tyLinkNtParamAlmData : REFERENCE TO tyAlmDat;
	p_tyLinkUsrMgmtAlmData : REFERENCE TO tyAlmDat;
	p_tyLinkBuffer1AlmData : REFERENCE TO tyAlmDat;
	p_tyLinkBuffer2AlmData : REFERENCE TO tyAlmDat;
	p_tyLinkBuffer3AlmData : REFERENCE TO tyAlmDat;
	p_tyLinkUSSMEMAAAlmData : REFERENCE TO tyAlmDat;
	p_tyLinkUSSMEMABAlmData : REFERENCE TO tyAlmDat;
	p_tyLinkUSSMEMA1AlmData : REFERENCE TO tyAlmDat;
	p_tyLinkUSSMEMA2AlmData : REFERENCE TO tyAlmDat;
	p_tyLinkUSSMEMA3AlmData : REFERENCE TO tyAlmDat;
	p_tyLinkDSSMEMA1AlmData : REFERENCE TO tyAlmDat;
	p_tyLinkDSSMEMA2AlmData : REFERENCE TO tyAlmDat;
	p_tyLinkDSSMEMA3AlmData : REFERENCE TO tyAlmDat;
	p_tyLinkInShutterAlmData : REFERENCE TO tyAlmDat;
	p_tyLinkOutShutterAlmData : REFERENCE TO tyAlmDat;
	p_tyLinkOutShutterAlmData3 : REFERENCE TO tyAlmDat;
	p_tyLinkOutShutterAlmData2 : REFERENCE TO tyAlmDat;
	p_tyLinkStopperAAlmData : REFERENCE TO tyAlmDat;
	p_tyLinkStopperBAlmData : REFERENCE TO tyAlmDat;
	p_tyLinkPshrConvAlmData : REFERENCE TO tyAlmDat;
	p_tyLinkMagConv1AlmData : REFERENCE TO tyAlmDat;
	p_tyLinkMagConv2AlmData : REFERENCE TO tyAlmDat;
	p_tyLinkMagConv3AlmData : REFERENCE TO tyAlmDat;
	p_tyLinkAWOpenAlmData : REFERENCE TO tyAlmDat;
	p_tyLinkAWOpenAlmData1 : REFERENCE TO tyAlmDat;
	p_tyLinkAWOpenAlmData2 : REFERENCE TO tyAlmDat;
	p_tyLinkAWOpenAlmData3 : REFERENCE TO tyAlmDat;
	p_tyLinkTravAlmData : REFERENCE TO tyAlmDat;
	p_tyLinkTravAlmData1 : REFERENCE TO tyAlmDat;
	p_tyLinkTravAlmData2 : REFERENCE TO tyAlmDat;
	p_tyLinkTravAlmData3 : REFERENCE TO tyAlmDat;
	p_tyLinkLifterBtmAlmData : REFERENCE TO tyAlmDat;
	p_tyLinkLifterBtmAlmData1 : REFERENCE TO tyAlmDat;
	p_tyLinkLifterBtmAlmData2 : REFERENCE TO tyAlmDat;
	p_tyLinkLifterBtmAlmData3 : REFERENCE TO tyAlmDat;
	p_tyLinkDIAlmData1 : REFERENCE TO tyAlmDat;
	p_tyLinkDIAlmData2 : REFERENCE TO tyAlmDat;
	p_tyLinkDIAlmData3 : REFERENCE TO tyAlmDat;
	p_tyLinkDIAlmData4 : REFERENCE TO tyAlmDat;
	p_tyLinkDIAlmData5 : REFERENCE TO tyAlmDat;
	p_tyLinkDIAlmData6 : REFERENCE TO tyAlmDat;
	p_tyLinkAGVAlmData1 : REFERENCE TO tyAlmDat;
	p_tyLinkAGVMag1AlmData : REFERENCE TO tyAlmDat;
	p_tyLinkAGVMag2AlmData : REFERENCE TO tyAlmDat;
	p_tyLinkAGVMag3AlmData : REFERENCE TO tyAlmDat;
	p_tyLinkHermesAlmData : REFERENCE TO tyAlmDat;
	p_tyLinkUSHermesAAlmData : REFERENCE TO tyAlmDat;
	p_tyLinkUSHermesAAlmData1 : REFERENCE TO tyAlmDat;
	p_tyLinkUSHermesAAlmData2 : REFERENCE TO tyAlmDat;
	p_tyLinkUSHermesAAlmData3 : REFERENCE TO tyAlmDat;
	p_tyLinkUSHermesAAlmData4 : REFERENCE TO tyAlmDat;
	p_tyLinkUSHermesAAlmData5 : REFERENCE TO tyAlmDat;
	p_tyLinkUSHermesAInfoData : REFERENCE TO tyAlmDat;
	p_tyLinkUSHermesBAlmData : REFERENCE TO tyAlmDat;
	p_tyLinkUSHermesBAlmData1 : REFERENCE TO tyAlmDat;
	p_tyLinkUSHermesBAlmData2 : REFERENCE TO tyAlmDat;
	p_tyLinkUSHermesBAlmData3 : REFERENCE TO tyAlmDat;
	p_tyLinkUSHermesBAlmData4 : REFERENCE TO tyAlmDat;
	p_tyLinkUSHermesBAlmData5 : REFERENCE TO tyAlmDat;
	p_tyLinkUSHermesBInfoData : REFERENCE TO tyAlmDat;
	p_tyLinkRmtHermesAlmData : REFERENCE TO tyAlmDat;
	p_tyLinkRmtHermesAlmData1 : REFERENCE TO tyAlmDat;
	p_tyLinkRmtHermesAlmData2 : REFERENCE TO tyAlmDat;
	p_tyLinkRmtHermesAlmData3 : REFERENCE TO tyAlmDat;
	p_tyLinkSvyHermesAlmData1 : REFERENCE TO tyAlmDat;
	p_tyLinkSvyHermesAlmData2 : REFERENCE TO tyAlmDat;
	p_tyLinkSvyHermesAlmData3 : REFERENCE TO tyAlmDat;
	p_tyLinkSvyHermesAlmData4 : REFERENCE TO tyAlmDat;
	p_tyLinkSvyHermesInfoData : REFERENCE TO tyAlmDat;
	p_tyLinkSvyHermesInfoData1 : REFERENCE TO tyAlmDat;
	p_tyLinkSvyHermesInfoData2 : REFERENCE TO tyAlmDat;
	p_tyLinkSvyHermesInfoData3 : REFERENCE TO tyAlmDat;
	p_tyLinkSvyHermesInfoData4 : REFERENCE TO tyAlmDat;
	p_tyLinkSvyHermesAlmData : REFERENCE TO tyAlmDat;
	p_tyLinkLFLeaderAlmData : REFERENCE TO tyAlmDat;
	p_tyLinkLFFollowerAlmData : REFERENCE TO tyAlmDat;
	p_tyLinkLFFollowerInfoData : REFERENCE TO tyAlmDat;
	p_tyLinkLFFollowerInfoData1 : REFERENCE TO tyAlmDat;
	p_tyLinkFollower1AlmData : REFERENCE TO tyAlmDat;
	p_tyLinkFollower1InfoData : REFERENCE TO tyAlmDat;
	p_tyLinkFollower1InfoData1 : REFERENCE TO tyAlmDat;
	p_tyLinkFollower2AlmData : REFERENCE TO tyAlmDat;
	p_tyLinkFollower2InfoData : REFERENCE TO tyAlmDat;
	p_tyLinkFollower2InfoData1 : REFERENCE TO tyAlmDat;
	p_tyLinkLCSMngRcpAlmData : REFERENCE TO tyAlmDat;
	p_tyLinkMcAlarmData : REFERENCE TO tyAlmDat;
	p_tyLinkLCSLFAlmData : REFERENCE TO tyAlmDat;
	p_tyLinkLCSLFInfoData : REFERENCE TO tyAlmDat;
	p_tyLinkOpsTravLifULAlmData : REFERENCE TO tyAlmDat;
	p_tyLinkOpsMagUL1AlmData : REFERENCE TO tyAlmDat;
	p_tyLinkOpsMagUL1AlmData1 : REFERENCE TO tyAlmDat;
	p_tyLinkOpsMagUL2AlmData : REFERENCE TO tyAlmDat;
	p_tyLinkOpsMagUL2AlmData1 : REFERENCE TO tyAlmDat;
	p_tyLinkOpsMagUL3AlmData : REFERENCE TO tyAlmDat;
	p_tyLinkOpsMagUL3AlmData1 : REFERENCE TO tyAlmDat;
	p_tyLinkOpsLifMagULAlmData : REFERENCE TO tyAlmDat;
	p_tyLinkOpsLifMagULAlmData1 : REFERENCE TO tyAlmDat;
	p_tyLinkOpsLifMagULAlmData2 : REFERENCE TO tyAlmDat;
	p_tyLinkOpsMagConvUL1AlmData : REFERENCE TO tyAlmDat;
	p_tyLinkOpsMagConvUL1AlmData1 : REFERENCE TO tyAlmDat;
	p_tyLinkOpsMagConvUL2AlmData : REFERENCE TO tyAlmDat;
	p_tyLinkOpsMagConvUL2AlmData1 : REFERENCE TO tyAlmDat;
	p_tyLinkOpsMagConvUL3AlmData : REFERENCE TO tyAlmDat;
	p_tyLinkOpsMagConvUL3AlmData1 : REFERENCE TO tyAlmDat;
	p_tyLinkMag1SelClampAlmData : REFERENCE TO tyAlmDat;
	p_tyLinkMag2SelClampAlmData : REFERENCE TO tyAlmDat;
	p_tyLinkMag3SelClampAlmData : REFERENCE TO tyAlmDat;
	p_tyLinkMag1SafetyBarAlmData : REFERENCE TO tyAlmDat;
	p_tyLinkMag2SafetyBarAlmData : REFERENCE TO tyAlmDat;
	p_tyLinkMag3SafetyBarAlmData : REFERENCE TO tyAlmDat;
	p_tyLinkMag1AWEngageAlmData : REFERENCE TO tyAlmDat;
	p_tyLinkMag2AWEngageAlmData : REFERENCE TO tyAlmDat;
	p_tyLinkMag3AWEngageAlmData : REFERENCE TO tyAlmDat;
	p_tyLinkMagAWOpen1AlmData : REFERENCE TO tyAlmDat;
	p_tyLinkMagAWOpen1AlmData1 : REFERENCE TO tyAlmDat;
	p_tyLinkMagAWOpen1AlmData2 : REFERENCE TO tyAlmDat;
	p_tyLinkMagAWOpen1AlmData3 : REFERENCE TO tyAlmDat;
	p_tyLinkMagAWOpen2AlmData : REFERENCE TO tyAlmDat;
	p_tyLinkMagAWOpen2AlmData1 : REFERENCE TO tyAlmDat;
	p_tyLinkMagAWOpen2AlmData2 : REFERENCE TO tyAlmDat;
	p_tyLinkMagAWOpen2AlmData3 : REFERENCE TO tyAlmDat;
	p_tyLinkMagAWOpen3AlmData : REFERENCE TO tyAlmDat;
	p_tyLinkMagAWOpen3AlmData1 : REFERENCE TO tyAlmDat;
	p_tyLinkMagAWOpen3AlmData2 : REFERENCE TO tyAlmDat;
	p_tyLinkMagAWOpen3AlmData3 : REFERENCE TO tyAlmDat;
	p_tyLinkUSSOT1AlmData : REFERENCE TO tyAlmDat;
	p_tyLinkUSSOT2AlmData : REFERENCE TO tyAlmDat;
	p_tyLinkUSSOT3AlmData : REFERENCE TO tyAlmDat;
	p_tyLinkDSSOT1AlmData : REFERENCE TO tyAlmDat;
	p_tyLinkDSSOT2AlmData : REFERENCE TO tyAlmDat;
	p_tyLinkDSSOT3AlmData : REFERENCE TO tyAlmDat;
	p_tyLinkAWPushOrPullerAlmData : REFERENCE TO tyAlmDat;
	p_tyLinkAWPushOrPullerAlmData1 : REFERENCE TO tyAlmDat;
	p_tyLinkAWPushOrPullerAlmData2 : REFERENCE TO tyAlmDat;
	p_tyLinkAWPushOrPullerAlmData3 : REFERENCE TO tyAlmDat;
	p_tyLinkMtrPshrAlmData : REFERENCE TO tyAlmDat;
	p_tyLinkTopEntStprAlmData : REFERENCE TO tyAlmDat;
	p_tyLinkTopMidStprAlmData : REFERENCE TO tyAlmDat;
	p_tyLinkTopExtStprAlmData : REFERENCE TO tyAlmDat;
	p_tyLinkBtmMidStprAlmData : REFERENCE TO tyAlmDat;
	p_tyLinkBtmExtStprAlmData : REFERENCE TO tyAlmDat;
	p_tyLinkTopEntStpr2AlmData : REFERENCE TO tyAlmDat;
	p_tyLinkTopMidStpr2AlmData : REFERENCE TO tyAlmDat;
	p_tyLinkTopExtStpr2AlmData : REFERENCE TO tyAlmDat;
	p_tyLinkBtmMidStpr2AlmData : REFERENCE TO tyAlmDat;
	p_tyLinkBtmExtStpr2AlmData : REFERENCE TO tyAlmDat;
	p_tyLinkInMagConvAlmData : REFERENCE TO tyAlmDat;
	p_tyLinkOutMagConvAlmData : REFERENCE TO tyAlmDat;
	p_tyLinkInMagConv2AlmData : REFERENCE TO tyAlmDat;
	p_tyLinkOutMagConv2AlmData : REFERENCE TO tyAlmDat;
	p_tyLinkLifterMagConvAlmData : REFERENCE TO tyAlmDat;
	p_tyLinkLifterMagConv2AlmData : REFERENCE TO tyAlmDat;
	p_tyLinkOpsInMagConvAlmData : REFERENCE TO tyAlmDat;
	p_tyLinkOpsOutMagConvAlmData : REFERENCE TO tyAlmDat;
	p_tyLinkLifter2AlmData : REFERENCE TO tyAlmDat;
	p_tyLinkLifter2AlmData1 : REFERENCE TO tyAlmDat;
	p_tyLinkLifter2AlmData2 : REFERENCE TO tyAlmDat;
	p_tyLinkLifter2AlmData3 : REFERENCE TO tyAlmDat;
	p_tyLinkOpsStprAlmData : REFERENCE TO tyAlmDat;
	p_tyLinkPPAlmData : REFERENCE TO tyAlmDat;
	p_tyLinkPPAlmData1 : REFERENCE TO tyAlmDat;
	p_tyLinkPPAlmData2 : REFERENCE TO tyAlmDat;
	p_tyLinkPPAlmData3 : REFERENCE TO tyAlmDat;
	p_tyLinkTCPAlmData : REFERENCE TO tyAlmDat;
	p_tyLinkTCPAlmData1 : REFERENCE TO tyAlmDat;
	p_tyLinkTCPAlmData2 : REFERENCE TO tyAlmDat;
	p_tyLinkTCPAlmData3 : REFERENCE TO tyAlmDat;
	p_tyLinkTCPTopAlmData : REFERENCE TO tyAlmDat;
	p_tyLinkTCPBtmAlmData : REFERENCE TO tyAlmDat;
	p_tyLinkAutoRcpAlmData : REFERENCE TO tyAlmDat;
END_VAR
(**)
VAR
	fbDlyTmr : TON := (PT:=T#5s);
	fbDeleteLogTmr : TON := (PT:=T#24h);
END_VAR
```

#### Act_Link.st - Change By Project
```iecst
(** 2019-01-07 **)
ACTION Act_Link:

	(*IF EDGEPOS(p_tyLinkUSSMEMA1AlmData.udiCode <> 0) THEN
		p_tyLinkUSSMEMA1AlmData.sProgNm	:= 'Mag1_1';
		p_tyLinkUSSMEMA1AlmData.sAlmMsg	:= 'Pushing Board Failed';
	END_IF

	IF EDGEPOS(p_tyLinkUSSMEMA2AlmData.udiCode <> 0) THEN
		p_tyLinkUSSMEMA2AlmData.sProgNm	:= 'Mag2_1';
		p_tyLinkUSSMEMA2AlmData.sAlmMsg	:= 'Pushing Board Failed';
	END_IF

	IF EDGEPOS(p_tyLinkUSSMEMA3AlmData.udiCode <> 0) THEN
		p_tyLinkUSSMEMA3AlmData.sProgNm	:= 'Mag3_1';
		p_tyLinkUSSMEMA3AlmData.sAlmMsg	:= 'Pushing Board Failed';
	END_IF

	IF EDGEPOS(p_tyLinkDSSMEMA1AlmData.udiCode <> 0) THEN
		p_tyLinkDSSMEMA1AlmData.sProgNm	:= 'Mag1_2';
		p_tyLinkDSSMEMA1AlmData.sAlmMsg	:= 'Pushing Board Failed';
	END_IF

	IF EDGEPOS(p_tyLinkDSSMEMA2AlmData.udiCode <> 0) THEN
		p_tyLinkDSSMEMA2AlmData.sProgNm	:= 'Mag2_2';
		p_tyLinkDSSMEMA2AlmData.sAlmMsg	:= 'Pushing Board Failed';
	END_IF

	IF EDGEPOS(p_tyLinkDSSMEMA3AlmData.udiCode <> 0) THEN
		p_tyLinkDSSMEMA3AlmData.sProgNm	:= 'Mag3_2';
		p_tyLinkDSSMEMA3AlmData.sAlmMsg	:= 'Pushing Board Failed';
	END_IF*)

	//Index 1 For Internal Use

	pa_tyAlmData[2]		:= p_tyLinkUsrFolderAlmData;
	pa_tyAlmData[3]		:= p_tyLinkLibVerAlmData;
	pa_tyAlmData[4]		:= p_tyLinkTimeAlmData;
	pa_tyAlmData[5]		:= p_tyLinkTimeAlmData1;
	pa_tyAlmData[6]		:= p_tyLinkHWInfoAlmData;
	pa_tyAlmData[7]		:= p_tyLinkProdRcpAlmData;
	pa_tyAlmData[8]		:= p_tyLinkMpProdRcpAlmData;
	pa_tyAlmData[9]		:= p_tyLinkMagRcpAlmData;
	pa_tyAlmData[10]	:= p_tyLinkMcParamAlmData;
	pa_tyAlmData[11]	:= p_tyLinkNtParamAlmData;
	pa_tyAlmData[12]	:= p_tyLinkUsrMgmtAlmData;
	pa_tyAlmData[13]	:= p_tyLinkBuffer1AlmData;
	pa_tyAlmData[14]	:= p_tyLinkBuffer2AlmData;
	pa_tyAlmData[15]	:= p_tyLinkBuffer3AlmData;
	pa_tyAlmData[16]	:= p_tyLinkUSSMEMAAAlmData;
	pa_tyAlmData[17]	:= p_tyLinkUSSMEMABAlmData;
	pa_tyAlmData[18]	:= p_tyLinkUSSMEMA1AlmData;
	pa_tyAlmData[19]	:= p_tyLinkUSSMEMA2AlmData;
	pa_tyAlmData[20]	:= p_tyLinkUSSMEMA3AlmData;
	pa_tyAlmData[21]	:= p_tyLinkDSSMEMA1AlmData;
	pa_tyAlmData[22]	:= p_tyLinkDSSMEMA2AlmData;
	pa_tyAlmData[23]	:= p_tyLinkDSSMEMA3AlmData;
	pa_tyAlmData[24]	:= p_tyLinkInShutterAlmData;
	pa_tyAlmData[25]	:= p_tyLinkOutShutterAlmData;
	pa_tyAlmData[26]	:= p_tyLinkStopperAAlmData;
	pa_tyAlmData[27]	:= p_tyLinkStopperBAlmData;
	pa_tyAlmData[28]	:= p_tyLinkPshrConvAlmData;
	pa_tyAlmData[29]	:= p_tyLinkMagConv1AlmData;
	pa_tyAlmData[30]	:= p_tyLinkMagConv2AlmData;
	pa_tyAlmData[31]	:= p_tyLinkMagConv3AlmData;
	pa_tyAlmData[32]	:= p_tyLinkAWOpenAlmData;
	pa_tyAlmData[33]	:= p_tyLinkAWOpenAlmData1;
	pa_tyAlmData[34]	:= p_tyLinkAWOpenAlmData2;
	pa_tyAlmData[35]	:= p_tyLinkAWOpenAlmData3;
	pa_tyAlmData[36]	:= p_tyLinkTravAlmData;
	pa_tyAlmData[37]	:= p_tyLinkTravAlmData1;
	pa_tyAlmData[38]	:= p_tyLinkTravAlmData2;
	pa_tyAlmData[39]	:= p_tyLinkTravAlmData3;
	pa_tyAlmData[40]	:= p_tyLinkLifterBtmAlmData;
	pa_tyAlmData[41]	:= p_tyLinkLifterBtmAlmData1;
	pa_tyAlmData[42]	:= p_tyLinkLifterBtmAlmData2;
	pa_tyAlmData[43]	:= p_tyLinkLifterBtmAlmData3;
	pa_tyAlmData[44]	:= p_tyLinkDIAlmData1;
	pa_tyAlmData[45]	:= p_tyLinkDIAlmData2;
	pa_tyAlmData[46]	:= p_tyLinkDIAlmData3;
	pa_tyAlmData[47]	:= p_tyLinkDIAlmData4;
	pa_tyAlmData[48]	:= p_tyLinkAGVMag1AlmData;
	pa_tyAlmData[49]	:= p_tyLinkAGVMag2AlmData;
	pa_tyAlmData[50]	:= p_tyLinkAGVMag3AlmData;
	pa_tyAlmData[51]	:= p_tyLinkHermesAlmData;
	pa_tyAlmData[52]	:= p_tyLinkUSHermesAAlmData;
	pa_tyAlmData[53]	:= p_tyLinkUSHermesAAlmData1;
	pa_tyAlmData[54]	:= p_tyLinkUSHermesAAlmData2;
	pa_tyAlmData[55]	:= p_tyLinkUSHermesAAlmData3;
	pa_tyAlmData[56]	:= p_tyLinkUSHermesAAlmData4;
	pa_tyAlmData[57]	:= p_tyLinkUSHermesAInfoData;
	pa_tyAlmData[58]	:= p_tyLinkUSHermesBAlmData;
	pa_tyAlmData[59]	:= p_tyLinkUSHermesBAlmData1;
	pa_tyAlmData[60]	:= p_tyLinkUSHermesBAlmData2;
	pa_tyAlmData[61]	:= p_tyLinkUSHermesBAlmData3;
	pa_tyAlmData[62]	:= p_tyLinkUSHermesBAlmData4;
	pa_tyAlmData[63]	:= p_tyLinkUSHermesBInfoData;
	pa_tyAlmData[64]	:= p_tyLinkRmtHermesAlmData;
	pa_tyAlmData[65]	:= p_tyLinkRmtHermesAlmData1;
	pa_tyAlmData[66]	:= p_tyLinkRmtHermesAlmData2;
	pa_tyAlmData[67]	:= p_tyLinkRmtHermesAlmData3;
	pa_tyAlmData[68]	:= p_tyLinkLFLeaderAlmData;
	pa_tyAlmData[69]	:= p_tyLinkLFFollowerAlmData;
	pa_tyAlmData[70]	:= p_tyLinkLFFollowerInfoData;
	pa_tyAlmData[71]	:= p_tyLinkLFFollowerInfoData1;
	pa_tyAlmData[72]	:= p_tyLinkFollower1AlmData;
	pa_tyAlmData[73]	:= p_tyLinkFollower1InfoData;
	pa_tyAlmData[74]	:= p_tyLinkFollower1InfoData1;
	pa_tyAlmData[75]	:= p_tyLinkFollower2AlmData;
	pa_tyAlmData[76]	:= p_tyLinkFollower2InfoData;
	pa_tyAlmData[77]	:= p_tyLinkFollower2InfoData1;
	pa_tyAlmData[78]	:= p_tyLinkLCSMngRcpAlmData;
	pa_tyAlmData[79]	:= p_tyLinkLCSLFAlmData;
	pa_tyAlmData[80]	:= p_tyLinkLCSLFInfoData;
	pa_tyAlmData[81]	:= p_tyLinkOpsTravLifULAlmData;
//	pa_tyAlmData[82]	:= p_tyLinkOpsMagUL1AlmData;
//	pa_tyAlmData[83]	:= p_tyLinkOpsMagUL1AlmData1;
//	pa_tyAlmData[84]	:= p_tyLinkOpsMagUL2AlmData;
//	pa_tyAlmData[85]	:= p_tyLinkOpsMagUL2AlmData1;
//	pa_tyAlmData[86]	:= p_tyLinkOpsMagUL3AlmData;
//	pa_tyAlmData[87]	:= p_tyLinkOpsMagUL3AlmData1;
	pa_tyAlmData[82]	:= p_tyLinkOpsLifMagULAlmData;
	pa_tyAlmData[83]	:= p_tyLinkOpsLifMagULAlmData1;
	pa_tyAlmData[84]	:= p_tyLinkOpsLifMagULAlmData2;

	pa_tyAlmData[88]	:= p_tyLinkOpsMagConvUL1AlmData;
	pa_tyAlmData[89]	:= p_tyLinkOpsMagConvUL1AlmData1;
	pa_tyAlmData[90]	:= p_tyLinkOpsMagConvUL2AlmData;
	pa_tyAlmData[91]	:= p_tyLinkOpsMagConvUL2AlmData1;
	pa_tyAlmData[92]	:= p_tyLinkOpsMagConvUL3AlmData;
	pa_tyAlmData[93]	:= p_tyLinkOpsMagConvUL3AlmData1;
	pa_tyAlmData[94]	:= p_tyLinkUSHermesAAlmData5;
	pa_tyAlmData[95]	:= p_tyLinkUSHermesBAlmData5;
	pa_tyAlmData[96]	:= p_tyLinkMcAlarmData;
	pa_tyAlmData[97]	:= p_tyLinkMag1SafetyBarAlmData;
	pa_tyAlmData[98]	:= p_tyLinkMag2SafetyBarAlmData;
	pa_tyAlmData[99]	:= p_tyLinkMag3SafetyBarAlmData;
	pa_tyAlmData[100]	:= p_tyLinkMag1AWEngageAlmData;
	pa_tyAlmData[101]	:= p_tyLinkMag2AWEngageAlmData;
	pa_tyAlmData[102]	:= p_tyLinkMag3AWEngageAlmData;
	pa_tyAlmData[103]	:= p_tyLinkMag1SafetyBarAlmData;
	pa_tyAlmData[104]	:= p_tyLinkMag2SafetyBarAlmData;
	pa_tyAlmData[105]	:= p_tyLinkMag3SafetyBarAlmData;
	pa_tyAlmData[106]	:= p_tyLinkMag1AWEngageAlmData;
	pa_tyAlmData[107]	:= p_tyLinkMag2AWEngageAlmData;
	pa_tyAlmData[108]	:= p_tyLinkMag3AWEngageAlmData;
	pa_tyAlmData[109]	:= p_tyLinkMagAWOpen1AlmData;
	pa_tyAlmData[110]	:= p_tyLinkMagAWOpen1AlmData1;
	pa_tyAlmData[111]	:= p_tyLinkMagAWOpen1AlmData2;
	pa_tyAlmData[112]	:= p_tyLinkMagAWOpen1AlmData3;
	pa_tyAlmData[113]	:= p_tyLinkMagAWOpen2AlmData;
	pa_tyAlmData[114]	:= p_tyLinkMagAWOpen2AlmData1;
	pa_tyAlmData[115]	:= p_tyLinkMagAWOpen2AlmData2;
	pa_tyAlmData[116]	:= p_tyLinkMagAWOpen2AlmData3;
	pa_tyAlmData[117]	:= p_tyLinkMagAWOpen3AlmData;
	pa_tyAlmData[118]	:= p_tyLinkMagAWOpen3AlmData1;
	pa_tyAlmData[119]	:= p_tyLinkMagAWOpen3AlmData2;
	pa_tyAlmData[120]	:= p_tyLinkMagAWOpen3AlmData3;
	pa_tyAlmData[121]	:= p_tyLinkMcAlarmData;
	pa_tyAlmData[122]	:= p_tyLinkUSSOT1AlmData;
	pa_tyAlmData[123]	:= p_tyLinkUSSOT2AlmData;
	pa_tyAlmData[124]	:= p_tyLinkUSSOT3AlmData;
	pa_tyAlmData[125]	:= p_tyLinkDSSOT1AlmData;
	pa_tyAlmData[126]	:= p_tyLinkDSSOT2AlmData;
	pa_tyAlmData[127]	:= p_tyLinkDSSOT3AlmData;
	pa_tyAlmData[128]	:= p_tyLinkMag1SelClampAlmData;
	pa_tyAlmData[129]	:= p_tyLinkMag2SelClampAlmData;
	pa_tyAlmData[130]	:= p_tyLinkMag3SelClampAlmData;
	pa_tyAlmData[131]	:= p_tyLinkAWPushOrPullerAlmData;
	pa_tyAlmData[132]	:= p_tyLinkAWPushOrPullerAlmData1;
	pa_tyAlmData[133]	:= p_tyLinkAWPushOrPullerAlmData2;
	pa_tyAlmData[134]	:= p_tyLinkAWPushOrPullerAlmData3;
	pa_tyAlmData[135]	:= p_tyLinkMtrPshrAlmData;
	pa_tyAlmData[136]	:= p_tyLinkAGVAlmData1;
	pa_tyAlmData[150]	:= p_tyLinkDIAlmData5;

	IF p_bNtParamProjMagConvLane1Prep AND p_bNtParamProjMagConvLane2Prep THEN
		pa_tyAlmData[167]	:= p_tyLinkOpsInMagConvAlmData;
		pa_tyAlmData[168]	:= p_tyLinkOpsOutMagConvAlmData;
	END_IF
	IF p_bNtParamProjMagConvLane1Prep THEN //customized
		pa_tyAlmData[151]	:= p_tyLinkTopEntStprAlmData; //MagConv Lane1
		pa_tyAlmData[152]	:= p_tyLinkTopMidStprAlmData;
		pa_tyAlmData[153]	:= p_tyLinkTopExtStprAlmData;
		pa_tyAlmData[154]	:= p_tyLinkBtmMidStprAlmData;
		pa_tyAlmData[155]	:= p_tyLinkBtmExtStprAlmData;
		pa_tyAlmData[161]	:= p_tyLinkInMagConvAlmData;
		pa_tyAlmData[162]	:= p_tyLinkOutMagConvAlmData;
		pa_tyAlmData[165]	:= p_tyLinkLifterMagConvAlmData;
	END_IF
	IF  p_bNtParamProjMagConvLane2Prep  THEN
		pa_tyAlmData[156]	:= p_tyLinkTopEntStpr2AlmData; //MagConv Lane2
		pa_tyAlmData[157]	:= p_tyLinkTopMidStpr2AlmData;
		pa_tyAlmData[158]	:= p_tyLinkTopExtStpr2AlmData;
		pa_tyAlmData[159]	:= p_tyLinkBtmMidStpr2AlmData;
		pa_tyAlmData[160]	:= p_tyLinkBtmExtStpr2AlmData;
		pa_tyAlmData[163]	:= p_tyLinkInMagConv2AlmData;
		pa_tyAlmData[164]	:= p_tyLinkOutMagConv2AlmData;
		pa_tyAlmData[166]	:= p_tyLinkLifterMagConv2AlmData;
	END_IF
	IF p_bNtParamProjLifter2Prep THEN
		pa_tyAlmData[169]	:= p_tyLinkLifter2AlmData;
		pa_tyAlmData[170]	:= p_tyLinkLifter2AlmData1;
		pa_tyAlmData[171]	:= p_tyLinkLifter2AlmData2;
		pa_tyAlmData[172]	:= p_tyLinkLifter2AlmData3;
	END_IF
	pa_tyAlmData[173]	:= p_tyLinkPPAlmData;
	pa_tyAlmData[174]	:= p_tyLinkPPAlmData1;
	pa_tyAlmData[175]	:= p_tyLinkPPAlmData2;
	pa_tyAlmData[176]	:= p_tyLinkPPAlmData3;
	pa_tyAlmData[177]	:= p_tyLinkDIAlmData6;
	pa_tyAlmData[178]	:= p_tyLinkOutShutterAlmData2;
	pa_tyAlmData[179]	:= p_tyLinkOutShutterAlmData3;
	IF p_bNTParamTCPAGVSigPrep THEN
		pa_tyAlmData[180]	:= p_tyLinkTCPAlmData;
		pa_tyAlmData[181]	:= p_tyLinkTCPAlmData1;
		pa_tyAlmData[182]	:= p_tyLinkTCPAlmData2;
		pa_tyAlmData[183]	:= p_tyLinkTCPAlmData3;
	END_IF
	IF p_bNtParamTCPScannerPrep THEN
		pa_tyAlmData[184]	:= p_tyLinkTCPTopAlmData;
		pa_tyAlmData[185]	:= p_tyLinkTCPBtmAlmData;
	END_IF

	pa_tyAlmData[186] := p_tyLinkSvyHermesAlmData;
	pa_tyAlmData[187] := p_tyLinkSvyHermesAlmData1;
	pa_tyAlmData[188] := p_tyLinkSvyHermesAlmData2;
	pa_tyAlmData[189] := p_tyLinkSvyHermesAlmData3;
	pa_tyAlmData[190] := p_tyLinkSvyHermesAlmData4;
	pa_tyAlmData[191] := p_tyLinkSvyHermesInfoData;
	pa_tyAlmData[192] := p_tyLinkSvyHermesInfoData1;
	pa_tyAlmData[193] := p_tyLinkSvyHermesInfoData2;
	pa_tyAlmData[194] := p_tyLinkSvyHermesInfoData3;
	pa_tyAlmData[195] := p_tyLinkSvyHermesInfoData4;

	IF p_bNtParamAutoRcpPrep THEN
		pa_tyAlmData[195] :=  p_tyLinkAutoRcpAlmData;
	END_IF
END_ACTION
```

#### Cyclic.st - Do Not Change!!!
```iecst
(** 2019-03-29 **)
PROGRAM _CYCLIC

	IF bInitialDone = FALSE THEN
		IF g_tyStartUp.bNtSettingsLoadDone = TRUE  THEN
			bInitialDone	:= TRUE;

			Act_Initial;
		END_IF

	ELSE
		Act_InputConfig;
		Act_Main;
		Act_OutputConfig;
		Act_Alarm;

	END_IF

END_PROGRAM
```

#### Act_Initial.st - Do Not Change!!!
```iecst
(** 2019-01-03 **)
ACTION Act_Initial:

	//Initial
	sStatTxt	:= a_sStatText[eStat];

	fbDirCreate1.sDevice	:= 'F';
	fbDirCreate1.sDirName	:= 'User';
	fbDirCreate1(bEn := FALSE);

	fbDirCreate2.sDevice	:= 'User';
	fbDirCreate2.sDirName	:= 'Alarm';
	fbDirCreate2(bEn := FALSE);

	fbFileAppend1.sDevice	:= 'Alarm';
	fbFileAppend1(bEn := FALSE);

	fbFileOldDel1.sDevice	:= 'Alarm';
	fbFileOldDel1.sPath		:= '';
	fbFileOldDel1.sKeyword	:= 'ALARM_';
	fbFileOldDel1(bEn := FALSE);

	fbFileRead1.sDevice		:= 'Alarm';
	fbFileRead1.sFile		:= 'History.dat';
	fbFileRead1.udiOffset	:= 0;
	fbFileRead1.p_Dest		:= ADR(a_tyHistoryList);
	fbFileRead1.udiLen		:= SIZEOF(a_tyHistoryList);
	fbFileRead1(bEn := FALSE);

	fbFileWrite1.sDevice	:= 'Alarm';
	fbFileWrite1.sFile		:= 'History.dat';
	fbFileWrite1.udiOffset	:= 0;
	fbFileWrite1.p_Src		:= ADR(a_tyHistoryList);
	fbFileWrite1.udiLen		:= SIZEOF(a_tyHistoryList);
	fbFileWrite1.udiOption	:= 0;
	fbFileWrite1(bEn := FALSE);

	tylocalAlm.Out.bInfo					:= FALSE ;
END_ACTION
```
